VAR
	_config: INT;
END_VAR
IF Execute THEN	
	_logger.Information(_message.Reset().Append('ChuckInLoadingPosition: ').Append(TO_STRING(LoadingPosition)).ToString());
	
	IsInLoadingPosition := LoadingPosition;
	_chuckInLoadingPositionCmd := FALSE;
END_IF
END_METHOD

PROPERTY DeviceID : STRING
GET
DeviceID := _deviceID;
END_GET
SET
_deviceID := DeviceID;
END_SET
END_PROPERTY

PROPERTY Family : DeviceFamily
GET
Family := _family;
END_GET
SET
_family := Family;
END_SET
END_PROPERTY

METHOD PROTECTED IsAlive
VAR_INPUT
END_VAR
_notifyIsAlive := TRUE;

IF _lifeTimeCount < 5 THEN
	_lifeTimeCount := _lifeTimeCount + 1;
ELSE
	_lifeTimeCount := 1;
END_IF
END_METHOD

METHOD MessageSchedulerBase
VAR_INPUT
END_VAR
IF _pulseGeneratorBase.Q THEN
	_pulseGeneratorBase(IN := FALSE, PT := T#10MS);
		
	CASE _itemSchedulerBase OF			
		0:  _deliverMessagesBase := EFeedbackMsgChuckBase.IsInLoadingPositionMsg;
			ioMessage := ' ';
			_itemSchedulerBase := 1;
			
		1: _deliverMessagesBase := EFeedbackMsgChuckBase.IsInLoadingPositionMsg;
			ioMessage := TO_STRING(IsInLoadingPosition);
			_itemSchedulerBase := 0;
	END_CASE
ELSE
	_pulseGeneratorBase(IN := TRUE, PT := T#100MS);		
END_IF


IF _pulseIsAliveGenerator.Q THEN
	_pulseIsAliveGenerator(IN := FALSE, PT := T#10MS);
		
	IsAlive();	
ELSE
	_pulseIsAliveGenerator(IN := TRUE, PT := T#1000MS);		
END_IF
END_METHOD

PROPERTY Name : STRING
GET
Name := _name;
END_GET
SET
_name := Name;
END_SET
END_PROPERTY

PROPERTY WaferSize : EWaferSize
GET
WaferSize := _waferSize;
END_GET
SET
_waferSize := WaferSize;
END_SET
END_PROPERTY

END_FUNCTION_BLOCK

// ---- PMShared/Hardware/Devices/Ffus/Astrofan/Astrofan612Ffu.TcPOU
{attribute 'OPC.UA.DA' := '1'}
FUNCTION_BLOCK Astrofan612Ffu EXTENDS FfuBase
VAR
	{attribute 'OPC.UA.DA' := '0'}
	_master : ModbusRtuMasterV2_KL6x22B;
	{attribute 'OPC.UA.DA' := '0'}
	_modbusErrorId : MODBUS_ERRORS;
	{attribute 'OPC.UA.DA' := '0'}
	Quantity : WORD := 1;
	{attribute 'OPC.UA.DA' := '0'}
	Id : BYTE := 1;
	{attribute 'OPC.UA.DA' := '0'}
	_config : Astrofan612FfuConfig;		
	{attribute 'OPC.UA.DA' := '0'}
	_deliverMessages : INT;
	
	StateMsg : STRING(255);
	IsAliveMsg : STRING(255);
	CurrentSpeedMsg : STRING(255);
	TemperatureMsg : STRING(255);
	WarningRaisedMsg : STRING(255) := BOOL_TO_STRING(FALSE);
	AlarmRaisedMsg : STRING(255) := BOOL_TO_STRING(FALSE);
	CustomMsg : STRING(255);
	
	{region 'Commands'}
	{attribute 'OPC.UA.DA' := '0'}
	_powerOn : BOOL;
	{attribute 'OPC.UA.DA' := '0'}
	_powerOff : BOOL;
	{attribute 'OPC.UA.DA' := '0'}
	_customCmd : BOOL;
	{attribute 'OPC.UA.DA' := '0'}			  		   
	_raisePropertiesCmd : BOOL;
	{attribute 'OPC.UA.DA' := '0'}
	_cmd : STRING;	 
	{endregion}		
	{attribute 'OPC.UA.DA' := '0'}
	_initDevice : BOOL;	
	{attribute 'OPC.UA.DA' := '0'}
	_itemScheduler : INT;	
	{attribute 'OPC.UA.DA' := '0'}
	_pulseGenerator : TON;	
	{attribute 'OPC.UA.DA' := '0'}
	_pulseTimeout : TON;		
	{attribute 'OPC.UA.DA' := '0'}
	_itemRaisedProperties : INT;	
	{attribute 'OPC.UA.DA' := '0'}
	_pulseIsAliveGenerator : TON;	
	{attribute 'OPC.UA.DA' := '0'}
	_execPulseGenerator : TON;
	{attribute 'OPC.UA.DA' := '0'}
	_pulseLoop : TON;
	{attribute 'OPC.UA.DA' := '0'}	
	_itemSubScheduler : INT;
	{attribute 'OPC.UA.DA' := '0'}
	_itemExecScheduler : INT;
	{attribute 'OPC.UA.DA' := '0'}
	_itemSubRaisedProperties : INT;
	{attribute 'OPC.UA.DA' := '0'}
	_itemFanSpeed : INT;
	{attribute 'OPC.UA.DA' := '0'}
	message : STRING;
	{attribute 'OPC.UA.DA' := '0'}
	_lifeTimeCount : UINT;
	{attribute 'OPC.UA.DA' := '0'}
	_notifyIsAlive : BOOL;
	{attribute 'OPC.UA.DA' := '0'}
	_readData : UINT;
	{attribute 'OPC.UA.DA' := '0'}
	_readHoldingData : UINT;
	{attribute 'OPC.UA.DA' := '0'}
	_writeData : UINT;
	{attribute 'OPC.UA.DA' := '0'}
	_cmdReadInput : BOOL;
	{attribute 'OPC.UA.DA' := '0'}
	_cmdReadHolding : BOOL;
	{attribute 'OPC.UA.DA' := '0'}
	_cmdWriteSingleRegister : BOOL;
	{attribute 'OPC.UA.DA' := '0'}
	_addressInput : STRING;
	{attribute 'OPC.UA.DA' := '0'}
	_addressHolding : STRING;
	{attribute 'OPC.UA.DA' := '0'}
	_addressWrite : STRING;
	{attribute 'OPC.UA.DA' := '0'}
	_currentSpeedPercent : UINT;
	{attribute 'OPC.UA.DA' := '0'}	
	_temperature : UINT;
	{attribute 'OPC.UA.DA' := '0'}
	_maxSpeed : UINT;
	{attribute 'OPC.UA.DA' := '0'}
	_setSpeedCmd : BOOL;
	{attribute 'OPC.UA.DA' := '0'}
	_fanMaxSpeedCmd : BOOL;
	{attribute 'OPC.UA.DA' := '0'}
	_fanActualSpeedCmd : BOOL;
    {attribute 'OPC.UA.DA' := '0'}
	_setSpeedPercent : UINT;
	{attribute 'OPC.UA.DA' := '0'}
	_doneScheduler : BOOL;
	{attribute 'OPC.UA.DA' := '0'}
	_doneRaised : BOOL;
	{attribute 'OPC.UA.DA' := '0'}	
	_pressure AT %I* : UINT;
	{attribute 'OPC.UA.DA' := '0'}		
	_alarmRaised : EventRaised;
	{attribute 'OPC.UA.DA' := '0'}			
	_warningRaised : EventRaised;
END_VAR

ReadInputRegister();
ReadHoldingRegister();
WriteSingleRegister();

// Init device
InitDevice();

// Check if it's still alive
IF _notifyIsAlive THEN
	IsAliveMsg := TO_STRING(_lifeTimeCount);
	_notifyIsAlive := FALSE;
END_IF

CASE _deliverMessages OF
	EFeedbackMsgAstrofan612.StateMsg :
		;
	EFeedbackMsgAstrofan612.StatusMsg :
		;
	EFeedbackMsgAstrofan612.CurrentSpeedMsg :
		CurrentSpeedMsg := TO_STRING(_currentSpeedPercent);
	EFeedbackMsgAstrofan612.TemperatureMsg :
		TemperatureMsg := TO_STRING(_temperature);
	EFeedbackMsgAstrofan612.WarningRaisedMsg :
		;
	EFeedbackMsgAstrofan612.AlarmRaisedMsg :
		;
	EFeedbackMsgAstrofan612.CustomMsg :
		;
END_CASE

SetSpeed(_setSpeedCmd, _setSpeedPercent);
RaisePropertiesChanged(_raisePropertiesCmd);
CustomCommand(_customCmd, _cmd);


IF _config.Loop.IsEnabled THEN
	LoopFanSpeed();
	WarningRaised();
	AlarmRaised();	
END_IF


IF (NOT _setSpeedCmd AND NOT _customCmd AND NOT _raisePropertiesCmd) THEN
	MessageScheduler();
END_IF

METHOD AlarmRaised
VAR
	alarmRaised : STRING := 'ALARM';
END_VAR
_AlarmRaised(DeviceName := THIS^._name,
				EventRaisedMsg := alarmRaised,
				EventTimerSetCriteria := _currentSpeedPercent > _config.Loop.FfuLoopAlarm.ThresholdPercent, 
				EventTimerSeconds := _config.Loop.FfuLoopAlarm.TimerSeconds,
				EventMsg => );
				
IF 	_AlarmRaised.EventMsg = alarmRaised THEN
	AlarmRaisedMsg := BOOL_TO_STRING(TRUE);
ELSE
	AlarmRaisedMsg := BOOL_TO_STRING(FALSE);
END_IF
END_METHOD

{attribute 'TcRpcEnable' := '1'}
(** Custom command **)
METHOD CustomCommand
VAR_INPUT
	Execute : BOOL;
	Cmd : STRING;
END_VAR
(*IF Execute THEN
	_logger.Information(_message.Reset(). Append(_config.Name).Append(' - Custom command : '). Append(Cmd).ToString());	
	
	_deliverMessages := EFeedbackMsgAstrofan612.CustomMsg;														
	
	_customCmd := FALSE;
END_IF*)
END_METHOD

METHOD FB_init : BOOL
VAR_INPUT
	bInitRetains : BOOL; // if TRUE, the retain variables are initialized (warm start / cold start)
	bInCopyCode : BOOL;  // if TRUE, the instance afterwards gets moved into the copy code (online change)
	Config : Astrofan612FfuConfig;
END_VAR
IF Config.IsEnabled THEN
	_config := Config;
	
	SUPER^._ffuConfig.Name := Config.Name;
	SUPER^._ffuConfig.DeviceID := Config.DeviceID;
	SUPER^._ffuConfig.IsEnabled := Config.IsEnabled;
	SUPER^._ffuConfig.LogLevel := Config.LogLevel;

	SUPER^.Name := Config.Name;
	SUPER^.DeviceID := Config.DeviceID;	
	THIS^.Family := DeviceFamily.Ffu;
		
	_Logger.Information(_message.Reset().Append('Init ').
							Append('{').Append(TO_STRING(THIS^.Family)).Append('} - ').
							Append('{').Append(TO_STRING(Config.Name)).Append('}').ToString());	
END_IF
END_METHOD

METHOD GetFanActualSpeed 
VAR
	AddressActualSpeed : STRING := '16#D010';	
	currentSpeedReal : UINT;
END_VAR
IF _pulseGenerator.Q THEN
	_pulseGenerator(IN := FALSE, PT := T#10MS);
		
	CASE _itemSubScheduler OF
		0 :	_cmdReadInput := TRUE;
			_addressInput:= AddressActualSpeed;	
			_itemSubScheduler := 1;
		
		1 : _deliverMessages := EFeedbackMsgAstrofan612.CurrentSpeedMsg;
			_currentSpeedPercent := REAL_TO_UINT (( _readData * 100.00) / 65536);
			_cmdReadInput := FALSE;
			_itemSubScheduler := 0;
			_doneScheduler := TRUE;
	END_CASE	
ELSE
	_pulseGenerator(IN := TRUE, PT := T#500MS);		
END_IF
END_METHOD

METHOD GetFanMaxSpeed 
VAR
	AddressMaxSpeed : STRING := '16#D119';
END_VAR
IF _pulseGenerator.Q THEN
		_pulseGenerator(IN := FALSE, PT := T#10MS);
			
		CASE _itemSubRaisedProperties OF
			0 :	_cmdReadHolding := TRUE;
				_addressHolding := AddressMaxSpeed;
				_itemSubRaisedProperties := 1;
			
			1 : _maxSpeed := _readHoldingData;
				_cmdReadHolding := FALSE;
				_itemSubRaisedProperties := 0;		
	
				_doneRaised := TRUE;					
		END_CASE
	ELSE
		_pulseGenerator(IN := TRUE, PT := T#500MS);		
END_IF
END_METHOD

METHOD GetFanTemperature 
VAR
	AddressTemperature : STRING := '16#D015';
END_VAR
IF _pulseGenerator.Q THEN
	_pulseGenerator(IN := FALSE, PT := T#10MS);
		
	CASE _itemSubScheduler OF
		0 :	_cmdReadInput := TRUE;
			_addressInput := AddressTemperature;
			_itemSubScheduler := 1;
		
		1 : _deliverMessages := EFeedbackMsgAstrofan612.TemperatureMsg;
			_temperature := _readData;
			_cmdReadInput := FALSE;
			_itemSubScheduler := 0;
			
			_doneScheduler:= TRUE ;			
	END_CASE	
ELSE
	_pulseGenerator(IN := TRUE, PT := T#500MS);		
END_IF
END_METHOD

METHOD InitDevice
IF NOT _initDevice THEN	
	_logger.Information(_message.Reset(). Append(_config.Name). Append(' - Init device').ToString());
	
	THIS^.SetDone();
	
	_setSpeedPercent := 50;
	_setSpeedCmd := TRUE;
	_initDevice := TRUE;	
END_IF
END_METHOD

METHOD PROTECTED IsAlive
_notifyIsAlive := TRUE;

IF _lifeTimeCount < 5 THEN
	_lifeTimeCount := _lifeTimeCount + 1;
ELSE
	_lifeTimeCount := 1;
END_IF
END_METHOD

METHOD LoopFanSpeed 
VAR_INPUT
END_VAR
VAR
	differentialPressure : UINT;
END_VAR
IF _pulseLoop.Q THEN
	_pulseLoop(IN := FALSE, PT := T#10MS);
	
	differentialPressure := (_pressure * 10)/32767;
	
	IF differentialPressure <=  _config.Loop.FfuPressureMinimumValuePa THEN
		_setSpeedPercent := TO_UINT(LIMIT (_config.Loop.FfuLoopSetSpeedLowerLimitPercent, (_setSpeedPercent + 10), 
								_config.Loop.FfuLoopSetSpeedHigherLimitPercent));
		_setSpeedCmd := TRUE;
	ELSIF differentialPressure >= _config.Loop.FfuPressureMaximumValuePa THEN
		_setSpeedPercent := TO_UINT(LIMIT (_config.Loop.FfuLoopSetSpeedLowerLimitPercent, ABS(_setSpeedPercent - 10), 
								_config.Loop.FfuLoopSetSpeedHigherLimitPercent));
		_setSpeedCmd := TRUE;
	ELSE
		_SetSpeedPercent := _config.Loop.FfuLoopStandardSetSpeed;
		_setSpeedCmd := TRUE;
	END_IF
ELSE
	_pulseLoop(IN := TRUE, PT := TO_TIME(_config.Loop.FfuLoopPressureTimerSeconds*1000));
END_IF
END_METHOD

METHOD MessageScheduler
CASE _itemScheduler OF		
	0:	GetFanTemperature();	
		IF _doneScheduler THEN 
            _itemScheduler := 1;
		END_IF		
		
	1: GetFanActualSpeed();
	    IF _doneScheduler THEN 
            _itemScheduler := 0;
		END_IF	
	
END_CASE

_doneScheduler := FALSE;
END_METHOD

{attribute 'TcRpcEnable' := '1'}
METHOD RaisePropertiesChanged
VAR_INPUT
	execute : BOOL;
END_VAR
IF execute THEN
	_raisePropertiesCmd := TRUE;
	
	IF _pulseGenerator.Q THEN
		_pulseGenerator(IN := FALSE, PT := T#10MS);
		CASE _itemRaisedProperties OF
			0:  _deliverMessages := EFeedbackMsgAstrofan612.CurrentSpeedMsg;
				_currentSpeedPercent := 0;	
				_itemRaisedProperties := 1;
						
			1:	_deliverMessages := EFeedbackMsgAstrofan612.TemperatureMsg;
				_temperature := 0;	
				_itemRaisedProperties := 10;							
			
			10: _raisePropertiesCmd := FALSE;				
				_itemRaisedProperties := 0;		
		END_CASE
	ELSE
		_pulseGenerator(IN := TRUE, PT := T#50MS);	
	END_IF
END_IF
END_METHOD

METHOD ReadHoldingRegister
_master.ReadRegs (
	UnitID:= Id,
	Quantity:= Quantity,
	MBAddr:= STRING_TO_WORD(_addressHolding),
	cbLength:= SIZEOF(_readHoldingData),  
	pMemoryAddr:= ADR(_readHoldingData),  
	AuxQuantity:= ,     
	AuxMBAddr:= , 
	AuxcbLength:= , 
	pAuxMemoryAddr:= , 
	Execute:= _cmdReadHolding,
	Timeout:= T#1S,
	BUSY=> , 
	Error=> ,
	ErrorId=> _modbusErrorId, 
	cbRead=> );
END_METHOD

METHOD ReadInputRegister
_master.ReadInputRegs(
	UnitID:= Id,        
	Quantity:= Quantity,
	MBAddr:= STRING_TO_WORD(_addressInput),   
	cbLength:= SIZEOF(_readData),  
	pMemoryAddr:= ADR(_readData),  
	AuxQuantity:= ,     
	AuxMBAddr:= , 
	AuxcbLength:= , 
	pAuxMemoryAddr:= , 
	Execute:= _cmdReadInput,
	Timeout:= T#1S,
	BUSY=> , 
	Error=> , 
	ErrorId=> _modbusErrorId, 
	cbRead=> );
END_METHOD

{attribute 'TcRpcEnable' := '1'}
METHOD PROTECTED SetSpeed 
VAR_INPUT
	execute : BOOL;
	speedPercent : UINT;
END_VAR
VAR
	addressSetSpeed : STRING := '16#D001' ;
	setSpeed: UINT;
END_VAR
IF Execute THEN	
	_setSpeedCmd := TRUE;	
	_setSpeedPercent := SpeedPercent;

	IF _execPulseGenerator.Q THEN
		_execPulseGenerator(IN := FALSE, PT := T#10MS);
			
		CASE _itemExecScheduler OF
			0: 	
				_cmdReadInput := FALSE;
				_cmdReadHolding := FALSE;	
				_cmdWriteSingleRegister := FALSE;				
				_itemExecScheduler := 1;
				
			1:	IF _config.SpeedMatrix.Enable THEN
					setSpeed := ScaleSpeed(iSpeed := _setSpeedPercent, SpeedMatrix := _config.SpeedMatrix.FfuMatrix);
				ELSE
					setSpeed := _setSpeedPercent;
				END_IF
				_writeData := ((setSpeed * 65535) / 100);
				
				 _addressWrite := AddressSetSpeed;
				 _cmdWriteSingleRegister := TRUE;
				 _itemExecScheduler := 10;				
											
			10:  _cmdWriteSingleRegister := FALSE;
				_itemExecScheduler := 11;
			
			11:	GetFanActualSpeed();
				// TODO :  intégrer une tempo pour sortir de là, en cas de problème. Pour éviter la boucle infinie
				IF _doneScheduler  THEN
					_itemExecScheduler := 50;
					_doneScheduler := FALSE;
				END_IF
				
			50:  _cmdReadInput := FALSE;				
				_setSpeedCmd := FALSE;	
				_itemExecScheduler := 0;										
		END_CASE						
	ELSE
		_execPulseGenerator(IN := TRUE, PT := T#200MS);	
	END_IF
END_IF
END_METHOD

METHOD WarningRaised 
VAR
	warningRaised : STRING := 'Warning';
END_VAR
_warningRaised(DeviceName := THIS^._name,
				EventRaisedMsg := warningRaised,
				EventTimerSetCriteria := _currentSpeedPercent > _config.Loop.FfuLoopWarning.ThresholdPercent, 
				EventTimerSeconds := _config.Loop.FfuLoopWarning.TimerSeconds,
				EventMsg => );



IF 	_warningRaised.EventMsg = warningRaised THEN
	WarningRaisedMsg :=  BOOL_TO_STRING(TRUE);
ELSE
	WarningRaisedMsg :=  BOOL_TO_STRING(FALSE);
END_IF
END_METHOD

METHOD WriteSingleRegister
_master.WriteSingleRegister (
	UnitID:= Id,        
	Quantity:= Quantity,
	MBAddr:= STRING_TO_WORD(_addressWrite),   
	cbLength:= SIZEOF(_writeData),  
	pMemoryAddr:= ADR(_writeData),  
	AuxQuantity:= ,     
	AuxMBAddr:= , 
	AuxcbLength:= , 
	pAuxMemoryAddr:= , 
	Execute:= _cmdWriteSingleRegister,
	Timeout:= T#1S,
	BUSY=> , 
	Error=> , 
	ErrorId=> _modbusErrorId, 
	cbRead=> );
END_METHOD

END_FUNCTION_BLOCK

// ---- PMShared/Hardware/Devices/Ffus/FfuBase.TcPOU
FUNCTION_BLOCK ABSTRACT FfuBase EXTENDS TExecution IMPLEMENTS IDevice
VAR_INPUT
END_VAR
VAR_OUTPUT
END_VAR
VAR
	{attribute 'OPC.UA.DA' := '0'}
	_name : STRING;
	{attribute 'OPC.UA.DA' := '0'}
	_deviceID : STRING;				
	{attribute 'OPC.UA.DA' := '0'}	
	_family : DeviceFamily;	
	{attribute 'OPC.UA.DA' := '0'}
	_logger : Logger;
	{attribute 'OPC.UA.DA' := '0'}
	_message : StringBuilder;
	{attribute 'OPC.UA.DA' := '0'}
	_ffuConfig : DeviceConfiguration;	
END_VAR

PROPERTY DeviceID : STRING
GET
DeviceID := _deviceID;
END_GET
SET
_deviceID := DeviceID;
END_SET
END_PROPERTY

PROPERTY Family : DeviceFamily
GET
Family := _family;
END_GET
SET
_family := Family;
END_SET
END_PROPERTY

PROPERTY Name : STRING
GET
Name := _name;
END_GET
SET
_name := Name;
END_SET
END_PROPERTY

METHOD PROTECTED ABSTRACT SetSpeed
VAR_INPUT
	Execute : BOOL;
	SpeedPercent : UINT;
END_VAR
END_METHOD

END_FUNCTION_BLOCK

// ---- PMShared/Hardware/Devices/Ffus/Astrofan/Loop/EventRaise/EventRaised.TcPOU
FUNCTION_BLOCK EventRaised
VAR_INPUT
	EventRaisedMsg : STRING;
	EventTimerSeconds : UINT;
	EventTimerSetCriteria : BOOL;
	DeviceName	: STRING;
END_VAR
VAR_OUTPUT
	EventMsg : STRING;
END_VAR
VAR
	_eventtrigger : BOOL := FALSE;
	{attribute 'OPC.UA.DA' := '0'}	
	_eventRaised : BOOL;
	{attribute 'OPC.UA.DA' := '0'}	
	_eventTimeOut : TON;
	{attribute 'OPC.UA.DA' := '0'}	
	_logger : Logger;
	{attribute 'OPC.UA.DA' := '0'}
	_message : StringBuilder;
END_VAR

_eventTimeOut(IN := EventTimerSetCriteria,
			PT := TO_TIME(EventTimerSeconds*1000));
	IF _eventTimeOut.Q THEN
		_eventRaised := TRUE;
		eventMsg := EventRaisedMsg;
		IF	NOT _eventtrigger THEN
			_Logger.Information(_message.Reset().Append(eventMsg).Append(' - ').Append(DeviceName).ToString()); 
			_Eventtrigger := TRUE;
		END_IF
	ELSE
		_eventtrigger := FALSE;
		_eventRaised := FALSE;
		eventMsg := '';
	END_IF

END_FUNCTION_BLOCK

// ---- PMShared/Hardware/Devices/Ffus/Astrofan/Loop/FfuSpeedMatrix/ScaleSpeed.TcPOU
FUNCTION ScaleSpeed : UINT
VAR_INPUT
	iSpeed : UINT;
	SpeedMatrix	: ARRAY[0..Constants.speedMatrixSize] OF FfuSpeed;
END_VAR
VAR
	i : UINT;
	found	: BOOL := FALSE;
END_VAR

FOR i:= 1 TO Constants.speedMatrixSize DO
	IF (SpeedMatrix[i].NonScaledSpeedValue = iSpeed) THEN
		ScaleSpeed := SpeedMatrix[i].ScaledSpeedValue;
		found := TRUE;
	EXIT;
	END_IF
END_FOR

IF NOT found THEN
	ScaleSpeed := 0;
END_IF

END_FUNCTION

// ---- PMShared/Hardware/Devices/Screens/Densitron/DM430GNS/DM430GNScreenFS.TcPOU
{attribute 'OPC.UA.DA' := '1'}
FUNCTION_BLOCK DM430GNScreenFS EXTENDS DM430GNScreen
VAR_INPUT
END_VAR
VAR_OUTPUT
END_VAR
VAR
	{attribute 'OPC.UA.DA' := '0'}
	_config : DM430GNScreenConfig;
	{attribute 'OPC.UA.DA' := '0'}
	_coeAccess : CoeAccess;
	{attribute 'OPC.UA.DA' := '0'}
	_initConfigSerialCom : BOOL;
	{attribute 'OPC.UA.DA' := '0'}	
	_serialCom  : SerialCom(Prefix :='', Suffix := Const.CARRIAGE_RETURN);
	{attribute 'OPC.UA.DA' := '0'}
	_refSerialCom : REFERENCE TO SerialCom(Prefix :='', Suffix := Const.CARRIAGE_RETURN) := _serialCom;	
	
	{attribute 'OPC.UA.DA' := '0'}
	_pulseGeneratorInit : TON;	
	{attribute 'OPC.UA.DA' := '0'}
	_itemInit : INT;
END_VAR

IF _config.IsSimulated THEN
	SUPER^(Conf := _config, SerialCom := _serialCom, RefSerialCom := _refSerialCom);
ELSE
	IF NOT InitConfigSerialCom THEN
		ConfigureSerialCom();
	ELSIF THIS^.Status = TExecutionState.Ready THEN
		IF _refSerialCom.ErrorReceiveId = COMERROR_NOERROR THEN
			_refSerialCom(TxBuffer:= HardwareGlobalVariables.TxBufferDM430GNScreenFS, 
						  RxBuffer:= HardwareGlobalVariables.RxBufferDM430GNScreenFS);
		END_IF						  			
					
		SUPER^(Conf := _config, SerialCom := _serialCom, RefSerialCom := _refSerialCom);

		// Init device
		InitDevice(); 			
	END_IF
END_IF

METHOD ConfigureSerialCom
VAR_INPUT
END_VAR

VAR
	Status: INT;
END_VAR
IF _coeAccess.CoeOperation.Ready THEN
	_logger.Information(_message.Reset().Append('Start configuration com serial').ToString());
END_IF;	

_coeAccess.CoeOperation.Start();
_coeAccess(SerialCommunication := _config.SerialCommunication);
	
IF _coeAccess.CoeOperation.Done THEN
	_coeAccess.SetDone();
	
	_Logger.Information(_message.Reset().
							Append('{').Append(TO_STRING(THIS^.Family)).Append('} : ').
							Append(' - Status : ').Append(TO_STRING(_coeAccess.Status)).ToString());
	InitConfigSerialCom := TRUE;
END_IF
 
IF _coeAccess.CoeOperation.Error THEN	
	_coeAccess.SetError(0);
	
	_Logger.Error(_message.Reset().
							Append('{').Append(TO_STRING(THIS^.Family)).Append('} : ').
							Append(' - Status : ').Append(TO_STRING(_coeAccess.Status)).ToString());
	InitConfigSerialCom := TRUE;
END_IF

THIS^.Status := _coeAccess.Status;
State := _coeAccess.Status;
END_METHOD

METHOD FB_init : BOOL
VAR_INPUT
	bInitRetains : BOOL; // if TRUE, the retain variables are initialized (warm start / cold start)
	bInCopyCode : BOOL;  // if TRUE, the instance afterwards gets moved into the copy code (online change)
	Config : DM430GNScreenConfig;
END_VAR
IF Config.IsEnabled THEN
	_config := Config;
	
	SUPER^._screenConfig.Name := Config.Name;
	SUPER^._screenConfig.DeviceID := Config.DeviceID;
	SUPER^._screenConfig.IsEnabled := Config.IsEnabled;
	SUPER^._screenConfig.LogLevel := Config.LogLevel;
	
	SUPER^.Name := Config.Name;
	SUPER^.DeviceID := Config.DeviceID;	
	THIS^.Family := DeviceFamily.Screen;
		
	_Logger.Information(_message.Reset().Append('Init ').
							Append('{').Append(TO_STRING(THIS^.Family)).Append('} - ').
							Append('{').Append(TO_STRING(Config.Name)).Append('}').ToString());																													
END_IF
END_METHOD

PROPERTY InitConfigSerialCom : BOOL
GET
InitConfigSerialCom := _initConfigSerialCom;
END_GET
SET
_initConfigSerialCom := InitConfigSerialCom;
END_SET
END_PROPERTY

METHOD InitDevice
VAR_INPUT
END_VAR
VAR	
END_VAR
IF NOT _initDevice THEN		
	IF _pulseGeneratorInit.Q THEN
		_pulseGeneratorInit(IN := FALSE, PT := T#10MS);
			
		CASE _itemInit OF
			0:  _logger.Information(_message.Reset().Append(_config.Name).Append(' - Start to on').ToString());		
				_itemInit := 1;
				
			1:  _initDevice := TRUE;
				_itemInit := 0;
		END_CASE
	ELSE
		_pulseGeneratorInit(IN := TRUE, PT := T#500MS);	
	END_IF
END_IF
END_METHOD

END_FUNCTION_BLOCK

// ---- PMShared/Hardware/Devices/Screens/Densitron/DM430GNScreen.TcPOU
{attribute 'OPC.UA.DA' := '1'}
FUNCTION_BLOCK DM430GNScreen EXTENDS ScreenBase
VAR_INPUT	
	{attribute 'OPC.UA.DA' := '0'}
	Conf : DM430GNScreenConfig;		
	{attribute 'OPC.UA.DA' := '0'}
	SerialCom  : SerialCom(Prefix :='', Suffix := Const.CARRIAGE_RETURN);
	{attribute 'OPC.UA.DA' := '0'}
	RefSerialCom : REFERENCE TO SerialCom(Prefix :='', Suffix := Const.CARRIAGE_RETURN) := SerialCom;	
END_VAR
VAR_OUTPUT
END_VAR
VAR	
	{attribute 'OPC.UA.DA' := '0'}
	_deliverMessages : INT;
	
	StateMsg : STRING(255);
	StatusMsg : STRING(255);
	IsAliveMsg : STRING(255);
	PowerStateMsg : STRING(255);
	BacklightMsg : STRING(255);
	BrightnessMsg : STRING(255);
	ContrastMsg : STRING(255);
	FanAutoMsg : STRING(255);
	FanStepMsg : STRING(255);
	FanRpmMsg : STRING(255);
	TemperatureMsg : STRING(255);	
	CustomMsg : STRING(255);
	
	{region 'Commands'}
	
	{attribute 'OPC.UA.DA' := '0'}
	_powerOn : BOOL;
	{attribute 'OPC.UA.DA' := '0'}
	_powerOff : BOOL;
	
	{attribute 'OPC.UA.DA' := '0'}
	_backlight : BOOL;
	{attribute 'OPC.UA.DA' := '0'}
	_brightness : BOOL;
	{attribute 'OPC.UA.DA' := '0'}
	_contrast : BOOL;
	{attribute 'OPC.UA.DA' := '0'}
	_defaultValue : BOOL;
	{attribute 'OPC.UA.DA' := '0'}
	_fanStep : BOOL;
	{attribute 'OPC.UA.DA' := '0'}
	_sharpness : BOOL;
	{attribute 'OPC.UA.DA' := '0'}
	_fanAuto : BOOL;
	{attribute 'OPC.UA.DA' := '0'}
	_fanAutoOnCmd : BOOL;
	{attribute 'OPC.UA.DA' := '0'}
	_customCmd : BOOL;
	{attribute 'OPC.UA.DA' := '0'}			  		   
	_raiseProperties : BOOL;
	{attribute 'OPC.UA.DA' := '0'}	 
	_restoreParameters : BOOL;
	{attribute 'OPC.UA.DA' := '0'}
	_cmd : STRING;
	{attribute 'OPC.UA.DA' := '0'}
	_screenOn : BOOL;
	{attribute 'OPC.UA.DA' := '0'}
	_setBacklight : UINT;
	{attribute 'OPC.UA.DA' := '0'}
	_setBrightness : UINT;
	{attribute 'OPC.UA.DA' := '0'}
	_setContrast : UINT;
	{attribute 'OPC.UA.DA' := '0'}
	_setFanStep : EDisplayControlStep;	
	{attribute 'OPC.UA.DA' := '0'}
	_setSharpness : EDisplayControlStep;		
	{attribute 'OPC.UA.DA' := '0'}
	_ioRelayActivated : BOOL; 
				   
	{attribute 'OPC.UA.DA' := '0'}
	_screenSide : STRING;
	{attribute 'OPC.UA.DA' := '0'}
	_side : STRING;
	{attribute 'OPC.UA.DA' := '0'}
	_delimeter : STRING := ';';
		 
	{endregion}		

	{attribute 'OPC.UA.DA' := '0'}
	_initDevice : BOOL;	
	
	{attribute 'OPC.UA.DA' := '0'}
	_itemScheduler : INT;	
	{attribute 'OPC.UA.DA' := '0'}
	_pulseGenerator : TON;	
	{attribute 'OPC.UA.DA' := '0'}
	_pulseTimeout : TON;			
	{attribute 'OPC.UA.DA' := '0'}
	_itemRaisedProperties : INT;
	{attribute 'OPC.UA.DA' := '0'}
	_itemRestoreParameters : INT;	
	{attribute 'OPC.UA.DA' := '0'}
	_pulseIsAliveGenerator : TON;
	{attribute 'OPC.UA.DA' := '0'}
	_execPulseGenerator : TON;		
	{attribute 'OPC.UA.DA' := '0'}
	_execItemScheduler : INT;
	
	{attribute 'OPC.UA.DA' := '0'}
	message : STRING;
	
	{attribute 'OPC.UA.DA' := '0'}
	_lifeTimeCount : UINT;
	{attribute 'OPC.UA.DA' := '0'}
	_notifyIsAlive : BOOL;
END_VAR

IF SerialCom.ErrorSendId <> COMERROR_NOERROR THEN
	RETURN;
END_IF 

// Check if it's still alive	
IF _notifyIsAlive THEN
	IsAliveMsg := TO_STRING(_lifeTimeCount);
	_notifyIsAlive := FALSE;
END_IF

// Deliver messages
IF RefSerialCom.IsReceived THEN
	IF (Conf.DeviceID = TO_STRING(EScreenSide.Front)) THEN
		_screenSide := TO_STRING(EScreenSide.Front);
	ELSE
		_screenSide := TO_STRING(EScreenSide.Back);
	END_IF
	
	_side := CONCAT(_screenSide, _delimeter);
	message := RefSerialCom.LastReceivedString;
	
	CASE _deliverMessages OF		
		EFeedbackMsgDM430GN.StateMsg :
			;			
		EFeedbackMsgDM430GN.StatusMsg :
			;			
		EFeedbackMsgDM430GN.PowerStateMsg :
			PowerStateMsg := CONCAT(_side, ExtractMessage(message));		
		EFeedbackMsgDM430GN.BacklightMsg :
			BacklightMsg := CONCAT(_side, ExtractMessage(message));
		EFeedbackMsgDM430GN.BrightnessMsg :
			BrightnessMsg := CONCAT(_side, ExtractMessage(message));
		EFeedbackMsgDM430GN.ContrastMsg :
			ContrastMsg := CONCAT(_side, ExtractMessage(message));
		EFeedbackMsgDM430GN.FanAutoMsg :
			FanAutoMsg := CONCAT(_side, ExtractMessage(message));
		EFeedbackMsgDM430GN.FanStepMsg :
			FanStepMsg := CONCAT(_side, ExtractMessage(message));
		EFeedbackMsgDM430GN.FanRpmMsg :
			FanRpmMsg := CONCAT(_side, ExtractMessage(message));
		EFeedbackMsgDM430GN.TemperatureMsg :
			TemperatureMsg := CONCAT(_side, ExtractMessage(message));
		EFeedbackMsgDM430GN.CustomMsg :
			CustomMsg := CONCAT(_side, ExtractMessage(message));
	END_CASE	
END_IF						   							   		
	
PowerOn(_powerOn);
PowerOff(_powerOff);
SetBacklight(_backlight, _setBacklight);
SetBrightness(_brightness, _setBrightness);
SetContrast(_contrast, _setContrast);
SetDefaultValue(_defaultValue);
SetFanStep(_fanStep, _setFanStep);
SetSharpness(_sharpness, _setSharpness);
FanAutoOn(_fanAuto, _fanAutoOnCmd);
CustomCommand(_customCmd, _cmd);
RaisePropertiesChanged(_raiseProperties);	
RestoreParameters(_restoreParameters, _screenOn, _setBacklight, _setBrightness, _setContrast, _setSharpness);

IF (NOT _powerOn AND NOT _powerOff AND NOT _backlight AND NOT _brightness AND NOT _contrast AND NOT _defaultValue
 	AND NOT _fanStep AND NOT _sharpness AND NOT _fanAuto AND NOT _customCmd AND NOT _raiseProperties AND NOT _restoreParameters) THEN	
	MessageScheduler();	
END_IF

METHOD PRIVATE ConvertDecString : STRING
VAR_INPUT
	Cmd : STRING;
	Value : BYTE;
END_VAR
VAR
	tmp : STRING; 	
END_VAR

tmp := BYTE_TO_STRING(Value);
IF LEN(tmp) = 1 THEN
	tmp := BYTE_TO_DECSTR(Value, 3);
ELSIF LEN(tmp) = 2 THEN
	tmp := BYTE_TO_DECSTR(Value, 3);				
END_IF

ConvertDecString := CONCAT(cmd, tmp);
END_METHOD

{attribute 'TcRpcEnable' := '1'}
(** Custom command **)
METHOD CustomCommand
VAR_INPUT
	Execute : BOOL;
	Cmd : STRING;
END_VAR
VAR
END_VAR
IF Execute THEN
	_logger.Information(_message.Reset().Append(Conf.Name).Append(' - Custom command : ').Append(Cmd).ToString());	
	_deliverMessages := EFeedbackMsgDM430GN.CustomMsg;	
	
	SerialCom.Send(Cmd);
	_customCmd := FALSE;
END_IF
END_METHOD

METHOD PRIVATE ExtractMessage : STRING
VAR_INPUT
	Data : STRING;
END_VAR
VAR
	separator : STRING(3) := ' = ';
	split : ARRAY[0..1] OF STRING(255);
	resultSplit : BOOL;	
END_VAR

resultSplit := FindAndSplit(pSeparator := ADR(separator), pSrcString := ADR(RefSerialCom.LastReceivedString), 
                            pLeftString := ADR(split[0]), nLeftSize := SIZEOF(split[0]), 
                            pRightString := ADR(split[1]), nRightSize := SIZEOF(split[1]),
                            bSearchFromRight := FALSE );
IF resultSplit THEN
	ExtractMessage := DELETE(split[1], 1, LEN(split[1]));
ELSE	
	ExtractMessage := DELETE(RefSerialCom.LastReceivedString, 1, LEN(RefSerialCom.LastReceivedString));
END_IF
END_METHOD

{attribute 'TcRpcEnable' := '1'}
METHOD PROTECTED FanAutoOn
VAR_INPUT
	Execute : BOOL;
	AutoOn : BOOL; //0: OFF, 1: ON
END_VAR
VAR
	fanAuto : STRING;
	cmd : STRING := '000FA';
	mode : STRING;
END_VAR
IF Execute THEN	
	_fanAuto:= TRUE;	
	
	CASE _itemScheduler OF
		0:  IF AutoOn THEN
				fanAuto := 'N'; // N
				mode := 'ON';
			ELSE
				fanAuto := 'F'; // F
				mode := 'OFF';
			END_IF	
	
			_logger.Information(_message.Reset().Append(Conf.Name).Append(' - FanAutoOn: ').Append(mode).ToString());			
			SerialCom.Send(CONCAT(cmd, fanAuto)); 			
			_itemScheduler := 1;
		
		1:  GetFanAuto();				
			_fanAuto := FALSE;	
			_itemScheduler := 0;							
	END_CASE
	
	
END_IF
END_METHOD

METHOD PROTECTED GetBacklight 
VAR_INPUT
END_VAR
VAR
	cmd : STRING := '000GKV';
END_VAR
_deliverMessages := EFeedbackMsgDM430GN.BacklightMsg;
SerialCom.Send(cmd);
END_METHOD

METHOD PROTECTED GetBrightness 
VAR_INPUT
END_VAR
VAR
	cmd : STRING := '000GBV'; 
END_VAR
_deliverMessages := EFeedbackMsgDM430GN.BrightnessMsg;
SerialCom.Send(cmd);
END_METHOD

METHOD PROTECTED GetContrast 
VAR_INPUT
END_VAR
VAR
	cmd : STRING := '000GCV';
END_VAR
_deliverMessages := EFeedbackMsgDM430GN.ContrastMsg;
SerialCom.Send(cmd);
END_METHOD

METHOD PROTECTED GetFanAuto 
VAR_INPUT
END_VAR
VAR
	cmd : STRING := '000GFA'; 
END_VAR
_deliverMessages := EFeedbackMsgDM430GN.FanAutoMsg;
SerialCom.Send(cmd);
END_METHOD

METHOD PROTECTED GetFanRpm 
VAR_INPUT
END_VAR
VAR
	cmd : STRING := '000GFR';
END_VAR
_deliverMessages := EFeedbackMsgDM430GN.FanRpmMsg;
SerialCom.Send(cmd);
END_METHOD

METHOD PROTECTED GetFanStep 
VAR_INPUT
END_VAR
VAR
	cmd : STRING := '000GFV'; 
END_VAR
_deliverMessages := EFeedbackMsgDM430GN.FanStepMsg;
SerialCom.Send(cmd);
END_METHOD

METHOD PROTECTED GetPowerState 
VAR_INPUT
END_VAR
VAR 
	cmd : STRING := '000GPV';
END_VAR
_deliverMessages := EFeedbackMsgDM430GN.PowerStateMsg;
SerialCom.Send(cmd);
END_METHOD

METHOD PROTECTED GetTemperature 
VAR_INPUT
END_VAR
VAR
	cmd : STRING := '000GTV';
END_VAR
_deliverMessages := EFeedbackMsgDM430GN.TemperatureMsg;
SerialCom.Send(cmd);
END_METHOD

METHOD InitDevice
VAR_INPUT
END_VAR
IF NOT _initDevice THEN	
	_logger.Information(_message.Reset(). Append(Conf.Name). Append(' - Init device').ToString());
	
	THIS^.SetDone();
	_initDevice := TRUE;	
END_IF
END_METHOD

METHOD PROTECTED IsAlive
VAR_INPUT
END_VAR
_notifyIsAlive := TRUE;

IF _lifeTimeCount < 5 THEN
	_lifeTimeCount := _lifeTimeCount + 1;
ELSE
	_lifeTimeCount := 1;
END_IF
END_METHOD

METHOD MessageScheduler
VAR_INPUT
END_VAR
IF _pulseGenerator.Q THEN
	_pulseGenerator(IN := FALSE, PT := T#10MS);
	
	CASE _itemScheduler OF					
		0:	GetTemperature(); 
			_itemScheduler := 1;

		1:	GetPowerState(); 
			_itemScheduler := 0;	

	END_CASE
ELSE
	_pulseGenerator(IN := TRUE, PT := T#2000MS);		
END_IF



IF _pulseIsAliveGenerator.Q THEN
	_pulseIsAliveGenerator(IN := FALSE, PT := T#10MS);
		
	IsAlive();	
ELSE
	_pulseIsAliveGenerator(IN := TRUE, PT := T#1000MS);		
END_IF
END_METHOD

{attribute 'TcRpcEnable' := '1'}
METHOD PROTECTED PowerOff
VAR_INPUT
	Execute : BOOL;
END_VAR
VAR
	cmd : STRING := '000KPF'; 
END_VAR
IF Execute THEN	
	_logger.Information(_message.Reset().Append(Conf.Name).Append(' - PowerOff').ToString());
	SerialCom.Send(cmd);
	
	_powerOff := FALSE;
END_IF
END_METHOD

{attribute 'TcRpcEnable' := '1'}
METHOD PROTECTED PowerOn
VAR_INPUT
	Execute : BOOL;
END_VAR
VAR 
	cmd : STRING := '000KPN';
END_VAR
IF Execute THEN	
	_powerOn := TRUE;	
	
	IF _execPulseGenerator.Q THEN
		_execPulseGenerator(IN := FALSE, PT := T#10MS);
		CASE _execItemScheduler OF
			0: _logger.Information(_message.Reset().Append(Conf.Name).Append(' - PowerOn').ToString());
				SerialCom.Send(cmd);
				
				_execItemScheduler := 1;
			
			1:  GetPowerState();
				_execItemScheduler := 2;
	
			2:	_powerOn := FALSE;
				_execItemScheduler := 0;							
		END_CASE
	ELSE
		_execPulseGenerator(IN := TRUE, PT := T#400MS);	
	END_IF		
END_IF
END_METHOD

{attribute 'TcRpcEnable' := '1'}
METHOD RaisePropertiesChanged
VAR_INPUT
	Execute : BOOL;
END_VAR
IF Execute THEN		
	_raiseProperties := TRUE;	
	
	IF _pulseGenerator.Q THEN
		_pulseGenerator(IN := FALSE, PT := T#10MS);
		
		CASE _itemRaisedProperties OF		
			0:  StateMsg := ' ';
				StatusMsg := ' ';
				BacklightMsg := ' ';
				BrightnessMsg := ' ';
				ContrastMsg := ' ';
				FanAutoMsg := ' ';				
				FanStepMsg := ' ';
				FanRpmMsg := ' ';				
				CustomMsg := ' ';
				
				_itemRaisedProperties := 10;											
			
			10 : GetBacklight();
				 _itemRaisedProperties := 11;
				 
			11 : GetBrightness();
				 _itemRaisedProperties := 12;
				 
			12 : GetContrast();
				 _itemRaisedProperties := 13;
				 
			13 : GetFanAuto();
				 _itemRaisedProperties := 14;
				
			14 : GetFanRpm();
				_itemRaisedProperties := 15;
				
			15:  GetFanStep();
				_itemRaisedProperties := 16;				
							
			16:  _logger.Information(_message.Reset().Append(Conf.Name).Append(' - RaisePropertiesChanged').ToString());
				_raiseProperties := FALSE;				
				_itemRaisedProperties := 0;
		END_CASE
	
	ELSE
		_pulseGenerator(IN := TRUE, PT := T#200MS);	
	END_IF		
END_IF
END_METHOD

{attribute 'TcRpcEnable' := '1'}
METHOD RestoreParameters	
VAR_INPUT
	Execute : BOOL;
	ScreenOn : BOOL; 
	BacklightValue : UINT;
	BrightnessValue : UINT;
	ContrastValue : UINT;
	SharpnessValue : EDisplayControlStep;
END_VAR
IF Execute THEN		
	_restoreParameters := TRUE;	
	
	CASE _itemRestoreParameters OF		
		0:  _logger.Information(_message.Reset().Append(Conf.Name).Append(' - Start RestoreParameters').ToString());
			_itemRestoreParameters := 10;	
	
		10:  _powerOn := TRUE;
			IF NOT _powerOn THEN
				_itemRestoreParameters := 11;
			END_IF																		
		
		11 : _backlight := TRUE;
			_setBacklight := BacklightValue;
			
			IF NOT _backlight THEN
				_itemRestoreParameters := 12;
			END_IF
			 
		12 : _brightness := TRUE;
			_setBrightness := BrightnessValue;
    
			IF NOT _brightness THEN
				_itemRestoreParameters := 13;
			END_IF
			 
		13 : _contrast := TRUE;
			_setContrast := ContrastValue;
    
			IF NOT _contrast THEN
				_itemRestoreParameters := 14;
			END_IF
			 
		14 : _sharpness := TRUE;
			_setSharpness := SharpnessValue;
    
			IF NOT _sharpness THEN
				_itemRestoreParameters := 20;
			END_IF													
						
		20:  _logger.Information(_message.Reset().Append(Conf.Name).Append(' - Finish RestoreParameters').ToString());
			_restoreParameters := FALSE;				
			_itemRestoreParameters := 0;
	END_CASE		
END_IF
END_METHOD

{attribute 'TcRpcEnable' := '1'}
METHOD PROTECTED SetBacklight
VAR_INPUT
	Execute : BOOL;
	Value : UINT;
END_VAR
VAR	
	cmd : STRING := '000SKV';
END_VAR
IF Execute THEN	
	_backlight := TRUE;	
	_setBacklight := Value;
	
	IF _execPulseGenerator.Q THEN
		_execPulseGenerator(IN := FALSE, PT := T#10MS);
		CASE _execItemScheduler OF
			0:  IF _setBacklight >= 0 OR _setBacklight <= 100 THEN
					_logger.Information(_message.Reset().Append(Conf.Name).Append(' - SetBacklight: ').Append(TO_STRING(_setBacklight)).ToString());																	
					SerialCom.Send(ConvertDecString(cmd, UINT_TO_BYTE(_setBacklight)));					
				ELSE
					_logger.Error(_message.Reset().Append(Conf.Name).Append(' - SetBacklight - Out of range : ').Append(TO_STRING(_setBacklight)).ToString());				
				END_IF
				
				_execItemScheduler := 1;
			
			1:  GetBacklight();
				_execItemScheduler := 2;
	
			2:	_backlight := FALSE;	
				_execItemScheduler := 0;							
		END_CASE
	ELSE
		_execPulseGenerator(IN := TRUE, PT := T#400MS);	
	END_IF										
END_IF
END_METHOD

{attribute 'TcRpcEnable' := '1'}
METHOD PROTECTED SetBrightness
VAR_INPUT
	Execute : BOOL;
	Value : UINT;
END_VAR
VAR
	cmd : STRING := '000SBV';
END_VAR
IF Execute THEN	
	_brightness := TRUE;
	
	_setBrightness := Value;
	
	IF _execPulseGenerator.Q THEN
		_execPulseGenerator(IN := FALSE, PT := T#10MS);
		CASE _execItemScheduler OF
			0:  IF _setBrightness >= 0 OR _setBrightness <= 100 THEN
					_logger.Information(_message.Reset().Append(Conf.Name).Append(' - SetBrightness: ').Append(TO_STRING(_setBrightness)).ToString());									
					SerialCom.Send(ConvertDecString(cmd, UINT_TO_BYTE(_setBrightness)));					
				ELSE
					_logger.Error(_message.Reset().Append(Conf.Name).Append(' - SetBrightness - Out of range : ').Append(TO_STRING(_setBrightness)).ToString());
				END_IF
				
				_execItemScheduler := 1;
			
			1:  GetBrightness();
				_execItemScheduler := 2;
				
			2:	_brightness := FALSE;	
				_execItemScheduler := 0;							
		END_CASE
	ELSE
		_execPulseGenerator(IN := TRUE, PT := T#400MS);	
	END_IF										
END_IF
END_METHOD

{attribute 'TcRpcEnable' := '1'}
METHOD PROTECTED SetContrast
VAR_INPUT
	Execute : BOOL;
	Value : UINT;
END_VAR
VAR
	cmd : STRING := '000SCV';
	tmp : STRING;
END_VAR
IF Execute THEN	
	_contrast := TRUE;
	_setContrast := Value;
	
	IF _execPulseGenerator.Q THEN
		_execPulseGenerator(IN := FALSE, PT := T#10MS);
		CASE _execItemScheduler OF
			0:  IF _setContrast >= 0 OR _setContrast <= 100 THEN
					_logger.Information(_message.Reset().Append(Conf.Name).Append(' - SetContrast: ').Append(TO_STRING(_setContrast)).ToString());													
					SerialCom.Send(ConvertDecString(cmd, UINT_TO_BYTE(_setContrast)));					
				ELSE
					_logger.Error(_message.Reset().Append(Conf.Name).Append(' - SetContrast - Out of range : ').Append(TO_STRING(_setContrast)).ToString());
				END_IF
				
				_execItemScheduler := 1;
			
			1:  GetContrast();	
				_execItemScheduler := 2;
			
			2:	_contrast := FALSE;	
				_execItemScheduler := 0;							
		END_CASE	
	ELSE
		_execPulseGenerator(IN := TRUE, PT := T#400MS);	
	END_IF								
END_IF
END_METHOD

{attribute 'TcRpcEnable' := '1'}
METHOD PROTECTED SetDefaultValue
VAR_INPUT
	Execute : BOOL;
END_VAR
VAR	
	cmd : STRING := '000DFT'; 
END_VAR
IF Execute THEN		
	_logger.Information(_message.Reset().Append(Conf.Name).Append(' - SetDefaultValue').ToString());	
	SerialCom.Send(cmd);	
	
	_defaultValue := FALSE;
END_IF
END_METHOD

{attribute 'TcRpcEnable' := '1'}
METHOD PROTECTED SetFanStep
VAR_INPUT
	Execute : BOOL;
	Value : EDisplayControlStep;
END_VAR
VAR
	cmd : STRING := '000SFV00';
END_VAR
IF Execute THEN	
	_fanStep := TRUE;
	_setFanStep := Value;
	
	IF _execPulseGenerator.Q THEN
		_execPulseGenerator(IN := FALSE, PT := T#10MS);
		CASE _execItemScheduler OF
			0: _logger.Information(_message.Reset().Append(Conf.Name).Append(' - SetFanStep: ').Append(TO_STRING(_setFanStep)).ToString());			
				SerialCom.Send(CONCAT(cmd, TO_STRING(_setFanStep)));				
				_execItemScheduler := 1;
			
			1:  GetFanStep();	
				_execItemScheduler := 2;
			
			2:	_fanStep := FALSE;	
				_execItemScheduler := 0;							
		END_CASE	
	ELSE
		_execPulseGenerator(IN := TRUE, PT := T#400MS);	
	END_IF						
END_IF
END_METHOD

{attribute 'TcRpcEnable' := '1'}
METHOD PROTECTED SetSharpness
VAR_INPUT
	Execute : BOOL;
	Value : EDisplayControlStep;
END_VAR
VAR
	cmd : STRING := '000SSV00';
END_VAR
IF Execute THEN		
	_sharpness := TRUE;
	_setSharpness := Value;
 
	IF _execPulseGenerator.Q THEN
		_execPulseGenerator(IN := FALSE, PT := T#10MS);
		CASE _execItemScheduler OF
			0: _logger.Information(_message.Reset().Append(Conf.Name).Append(' - SetSharpness: ').Append(TO_STRING(_setSharpness)).ToString());
				SerialCom.Send(CONCAT(cmd, TO_STRING(_setSharpness)));				
				_execItemScheduler := 1;
			
			1:  _sharpness := FALSE;
				_execItemScheduler := 0;												
		END_CASE
	ELSE
		_execPulseGenerator(IN := TRUE, PT := T#400MS);	
	END_IF
END_IF
END_METHOD

END_FUNCTION_BLOCK

// ---- PMShared/Hardware/Devices/Screens/ScreenBase.TcPOU
FUNCTION_BLOCK ScreenBase EXTENDS TExecution IMPLEMENTS IDevice
VAR_INPUT
END_VAR
VAR_OUTPUT
END_VAR
VAR
	{attribute 'OPC.UA.DA' := '0'}
	_name : STRING;
	{attribute 'OPC.UA.DA' := '0'}
	_deviceID : STRING;				
	{attribute 'OPC.UA.DA' := '0'}	
	_family : DeviceFamily;	
	{attribute 'OPC.UA.DA' := '0'}
	_logger : Logger;
	{attribute 'OPC.UA.DA' := '0'}
	_message : StringBuilder;
	{attribute 'OPC.UA.DA' := '0'}
	_screenConfig : DeviceConfiguration;	
END_VAR

PROPERTY DeviceID : STRING
GET
DeviceID := _deviceID;
END_GET
SET
_deviceID := DeviceID;
END_SET
END_PROPERTY

PROPERTY Family : DeviceFamily
GET
Family := _family;
END_GET
SET
_family := Family;
END_SET
END_PROPERTY

PROPERTY Name : STRING
GET
Name := _name;
END_GET
SET
_name := Name;
END_SET
END_PROPERTY

END_FUNCTION_BLOCK

// ---- PMShared/Hardware/Devices/Screens/Densitron/DM430GNS/DM430GNScreenBS.TcPOU
{attribute 'OPC.UA.DA' := '1'}
FUNCTION_BLOCK DM430GNScreenBS EXTENDS DM430GNScreen
VAR_INPUT
END_VAR
VAR_OUTPUT
END_VAR
VAR
	{attribute 'OPC.UA.DA' := '0'}
	_config : DM430GNScreenConfig;
	{attribute 'OPC.UA.DA' := '0'}
	_coeAccess : CoeAccess;
	{attribute 'OPC.UA.DA' := '0'}
	_initConfigSerialCom : BOOL;
	{attribute 'OPC.UA.DA' := '0'}	
	_serialCom  : SerialCom(Prefix :='', Suffix := Const.CARRIAGE_RETURN);
	{attribute 'OPC.UA.DA' := '0'}
	_refSerialCom : REFERENCE TO SerialCom(Prefix :='', Suffix := Const.CARRIAGE_RETURN) := _serialCom;	
	
	{attribute 'OPC.UA.DA' := '0'}
	_pulseGeneratorInit : TON;	
	{attribute 'OPC.UA.DA' := '0'}
	_itemInit : INT;
END_VAR

IF _config.IsSimulated THEN
	SUPER^(Conf := _config, SerialCom := _serialCom, RefSerialCom := _refSerialCom);
ELSE
	IF NOT InitConfigSerialCom THEN
		ConfigureSerialCom();
	ELSIF THIS^.Status = TExecutionState.Ready THEN
		IF _refSerialCom.ErrorReceiveId = COMERROR_NOERROR THEN
			_refSerialCom(TxBuffer:= HardwareGlobalVariables.TxBufferDM430GNScreenBS, 
						  RxBuffer:= HardwareGlobalVariables.RxBufferDM430GNScreenBS);
		END_IF						  			
					
		SUPER^(Conf := _config, SerialCom := _serialCom, RefSerialCom := _refSerialCom);

		// Init device
		InitDevice(); 			
	END_IF
END_IF

METHOD ConfigureSerialCom
VAR_INPUT
END_VAR

VAR
	Status: INT;
END_VAR
IF _coeAccess.CoeOperation.Ready THEN
	_logger.Information(_message.Reset().Append('Start configuration com serial').ToString());
END_IF;	

_coeAccess.CoeOperation.Start();
_coeAccess(SerialCommunication := _config.SerialCommunication);
	
IF _coeAccess.CoeOperation.Done THEN
	_coeAccess.SetDone();
	
	_Logger.Information(_message.Reset().
							Append('{').Append(TO_STRING(THIS^.Family)).Append('} : ').
							Append(' - Status : ').Append(TO_STRING(_coeAccess.Status)).ToString());
	InitConfigSerialCom := TRUE;
END_IF
 
IF _coeAccess.CoeOperation.Error THEN	
	_coeAccess.SetError(0);
	
	_Logger.Error(_message.Reset().
							Append('{').Append(TO_STRING(THIS^.Family)).Append('} : ').
							Append(' - Status : ').Append(TO_STRING(_coeAccess.Status)).ToString());
	InitConfigSerialCom := TRUE;
END_IF

THIS^.Status := _coeAccess.Status;
State := _coeAccess.Status;
END_METHOD

METHOD FB_init : BOOL
VAR_INPUT
	bInitRetains : BOOL; // if TRUE, the retain variables are initialized (warm start / cold start)
	bInCopyCode : BOOL;  // if TRUE, the instance afterwards gets moved into the copy code (online change)
	Config : DM430GNScreenConfig;
END_VAR
IF Config.IsEnabled THEN
	_config := Config;
	
	SUPER^._screenConfig.Name := Config.Name;
	SUPER^._screenConfig.DeviceID := Config.DeviceID;
	SUPER^._screenConfig.IsEnabled := Config.IsEnabled;
	SUPER^._screenConfig.LogLevel := Config.LogLevel;
	
	SUPER^.Name := Config.Name;
	SUPER^.DeviceID := Config.DeviceID;	
	THIS^.Family := DeviceFamily.Screen;
		
	_Logger.Information(_message.Reset().Append('Init ').
							Append('{').Append(TO_STRING(THIS^.Family)).Append('} - ').
							Append('{').Append(TO_STRING(Config.Name)).Append('}').ToString());																													
END_IF
END_METHOD

PROPERTY InitConfigSerialCom : BOOL
GET
InitConfigSerialCom := _initConfigSerialCom;
END_GET
SET
_initConfigSerialCom := InitConfigSerialCom;
END_SET
END_PROPERTY

METHOD InitDevice
VAR_INPUT
END_VAR
VAR	
END_VAR
IF NOT _initDevice THEN		
	IF _pulseGeneratorInit.Q THEN
		_pulseGeneratorInit(IN := FALSE, PT := T#10MS);
			
		CASE _itemInit OF
			0:  _logger.Information(_message.Reset().Append(_config.Name).Append(' - Start to on').ToString());		
				_itemInit := 1;
							
			1:  _initDevice := TRUE;
				_itemInit := 0;
		END_CASE
	ELSE
		_pulseGeneratorInit(IN := TRUE, PT := T#500MS);	
	END_IF
END_IF
END_METHOD

END_FUNCTION_BLOCK

// ---- PMShared/Hardware/Devices/Rfids/Balluff/BisL405Rfid.TcPOU
{attribute 'OPC.UA.DA' := '1'}
FUNCTION_BLOCK BisL405Rfid EXTENDS RfidBase
VAR_INPUT
	IoBisL405Rfid : IoBisL405Rfid;
END_VAR
VAR_OUTPUT
END_VAR
VAR
	
	{attribute 'OPC.UA.DA' := '0'}
	_config : BisL405RfidConfig;
	
	{attribute 'OPC.UA.DA' := '0'}
	_deliverMessages : INT;
	
	DataCarrierMsg : STRING(255);
	
	{attribute 'OPC.UA.DA' := '0'}
	_initDevice : BOOL;
	
	{attribute 'OPC.UA.DA' := '0'}
	_itemInit : INT;
	
	{attribute 'OPC.UA.DA' := '0'}
	_itemScheduler : INT;
	{attribute 'OPC.UA.DA' := '0'}
	_itemExecScheduler : INT;
	
	{attribute 'OPC.UA.DA' := '0'}
	_itemExecReadTag : INT; //COUNTER
	{attribute 'OPC.UA.DA' := '0'}
	_itemExecReadTagWAIT : INT; //COUNTER
	
	{region ' CONFIGURE read BEHAVIOUR TEST options'}

	{attribute 'OPC.UA.DA' := '0'}
	_iReadTagTestRereadN : INT := 0; //3; number of time to re-read tag //CONFIGURE TEST //TEST ONLY

	{endregion}

	{region ' CONFIGURE read BEHAVIOUR options'}

	{attribute 'OPC.UA.DA' := '0'}
	_iReadStepMax : INT := 40; //max ticks/steps when tag detected //CONFIGURE 
	{attribute 'OPC.UA.DA' := '0'}
	_iReadStepMaxWait : INT := 10; //max ticks/steps when tag NOT detected //CONFIGURE 
	{attribute 'OPC.UA.DA' := '0'}
	_iReadTagBadFormatRereadN : INT := 3; //number of time to re-read tag (if 'TagBadFormat') //CONFIGURE 

	{endregion}

	{region 'control ACTIONS for signal input/output'}
	
	{attribute 'OPC.UA.DA' := '0'}
	_iDoReset : INT := 3;// 1=do it, >1 = COUNTDOWN //CONFIGURE restart at start of read
	{attribute 'OPC.UA.DA' := '0'}
	_iToggleAddressCountAfterReset : INT := 1; //3;// 1=do it, >1 = COUNTDOWN //CONFIGURE ---------------------------------------
	{attribute 'OPC.UA.DA' := '0'}
	_iToggleAddressCountAfterToggle : INT := 3;// 1=do it, >1 = COUNTDOWN //CONFIGURE -------------------------------------------
	{attribute 'OPC.UA.DA' := '0'}
	_iToggleAddress : INT := 0;// 1=do it, >1 = COUNTDOWN //CONFIGURE or set after 'Reset'/'Toggle'
	
	{attribute 'OPC.UA.DA' := '0'}
	_iReadTagRetry : INT := 0; //COUNT
	{attribute 'OPC.UA.DA' := '0'}
	_iReadDone : INT := 0; //COUNT
	{attribute 'OPC.UA.DA' := '0'}
	ToggleReset : BOOL;// := FALSE;//action flag
	{attribute 'OPC.UA.DA' := '0'}
	_uBitFlagWaitOn : UINT;// bit values 1=wait next 't' on, 2=wait 'S' on, 
	
	{attribute 'OPC.UA.DA' := '0'}
	_bPrevStrobe : BOOL;//save flag
	{attribute 'OPC.UA.DA' := '0'}
	_bLatchStrobeChanged : BOOL;//detect & latch
	{attribute 'OPC.UA.DA' := '0'}
	_bLatchADRToggled : BOOL := FALSE;//detect & latch
	
	{endregion}
	
	{attribute 'OPC.UA.DA' := '0'}
	_itemRaisedProperties : INT;
	{attribute 'OPC.UA.DA' := '0'}
	_pulseGenerator : TON;
	{attribute 'OPC.UA.DA' := '0'}
	_execPulseGenerator : TON;	
	
	{region 'Commands'}
	
	{attribute 'OPC.UA.DA' := '0'}			  		   
	_readTagCmd : BOOL;
	{attribute 'OPC.UA.DA' := '0'}			  		   
	_raiseProperties : BOOL;
	
	{endregion}	
	
	{attribute 'OPC.UA.DA' := '0'}
	message : STRING;
	
	{attribute 'OPC.UA.DA' := '0'}	
	_sMsgBuild : STRING;
END_VAR


// Init device
InitDevice(); 				  				 

// Deliver messages
CASE _deliverMessages OF			
	EFeedbackMsgBisL405.DataCarrierMsg :
		IF DataCarrierMsg <> message THEN
			DataCarrierMsg := message;	
		END_IF				
END_CASE							   							   	
	
ReadTag(_readTagCmd);
RaisePropertiesChanged(_raiseProperties);

IF NOT _raiseProperties THEN
	MessageScheduler();
END_IF

METHOD FB_init : BOOL
VAR_INPUT
	bInitRetains : BOOL; // if TRUE, the retain variables are initialized (warm start / cold start)
	bInCopyCode : BOOL;  // if TRUE, the instance afterwards gets moved into the copy code (online change)
	Config : BisL405RfidConfig;
END_VAR
IF Config.IsEnabled THEN
	_config := Config;
	
	SUPER^._rfidConfig.Name := Config.Name;
	SUPER^._rfidConfig.DeviceID := Config.DeviceID;
	SUPER^._rfidConfig.IsEnabled := Config.IsEnabled;
	SUPER^._rfidConfig.LogLevel := Config.LogLevel;
	
	SUPER^.Name := Config.Name;
	SUPER^.DeviceID := Config.DeviceID;
	
	THIS^.Family := DeviceFamily.Rfid;

	THIS^.SetReady();
	_Logger.Information(_message.Reset().Append('Init ').
							Append('{').Append(TO_STRING(THIS^.Family)).Append('} - ').
							Append('{').Append(TO_STRING(THIS^.Name)).Append('} - ').
							Append('Status : ').Append(TO_STRING(THIS^.Status)).
							ToString());										 
END_IF
END_METHOD

METHOD InitDataRead : BOOL
VAR_INPUT
END_VAR
//:	_sDBMsg:= '';//TEST ONLY
message := ' '; //clear result
_sMsgBuild := ' '; //clear result build
_itemExecReadTag := 0;//Reset read data step count
_itemExecReadTagWAIT := 0;//Reset read data step count
_iDoReset := 1;//do restart before read
_iToggleAddress:= 0;//INIT: //OFF
_uBitFlagWaitOn := 0;//INIT: 'DoReset' will set to 1 to wait for 't' signal (tag present)
_bLatchStrobeChanged:=TRUE; //INIT: bStrobeChange TRUE, set true for 1st 'ToggleAddress'
_bLatchADRToggled:=FALSE; //INIT: clear
END_METHOD

METHOD InitDevice
VAR_INPUT
END_VAR
IF NOT _initDevice THEN			
	_logger.Information(_message.Reset().
								Append(_config.Name).
								Append(' - init device').ToString());		
								
	_initDevice := TRUE;
END_IF
END_METHOD

METHOD MessageScheduler
VAR_INPUT
END_VAR
IF _pulseGenerator.Q THEN
	_pulseGenerator(IN := FALSE, PT := T#10MS);
		
	CASE _itemScheduler OF	
		0:	
			_itemScheduler := 10;
			
		10 : 
			_itemScheduler := 0;											
	END_CASE
ELSE
	_pulseGenerator(IN := TRUE, PT := T#100MS);	
END_IF
END_METHOD

{attribute 'TcRpcEnable' := '1'}
METHOD RaisePropertiesChanged
VAR_INPUT
	Execute : BOOL;
END_VAR
IF Execute THEN		
	_raiseProperties := TRUE;	
	
	IF _pulseGenerator.Q THEN
		_pulseGenerator(IN := FALSE, PT := T#10MS);
		
		CASE _itemRaisedProperties OF		
			0:  _readTagCmd := TRUE;
				_itemRaisedProperties := 10;
				
			10: _logger.Information(_message.Reset().Append(_config.Name).Append(' - RaisePropertiesChanged').ToString());
				_raiseProperties := FALSE;
				_itemRaisedProperties := 0;
		
		END_CASE
	
	ELSE
		_pulseGenerator(IN := TRUE, PT := T#100MS);	
	END_IF
		
END_IF
END_METHOD

{attribute 'TcRpcEnable' := '1'}
METHOD ReadTag
VAR_INPUT
	Execute : BOOL;
END_VAR
VAR
	CombinedByte: BYTE; 
	CombinedByte1: BYTE;

	bStrobeChange : BOOL;//detect
	//
	bLatchStrobeChanged : BOOL;//detect & latch, temp local copy...
	lRand:LREAL; //EC//20240715
	
	bTagValid : BOOL;
	
	lenghtMsg : INT;
END_VAR
IF Execute THEN
	_readTagCmd := TRUE;
	
	_deliverMessages := EFeedbackMsgBisL405.DataCarrierMsg;
	
	IF _execPulseGenerator.Q THEN
		_execPulseGenerator(IN := FALSE, PT := T#100MS);
			
		CASE _itemExecScheduler OF
			0:  //init for read
				_logger.Information(_message.Reset().Append(_config.Name).Append(' - ReadTag').ToString());
				_itemExecScheduler := 1;
				InitDataRead();
				SignalClear_ADR_and_RESTART();//clear at START
			
			1:  //reset reader & read tag data, byte by byte
				IF IoBisL405Rfid.Strobe <> _bPrevStrobe THEN
					bStrobeChange:=TRUE;
				ELSE
					bStrobeChange:=FALSE;
				END_IF
				_bPrevStrobe:= IoBisL405Rfid.Strobe;
				IF bStrobeChange THEN
					_bLatchStrobeChanged:=TRUE;//reset by 'ToggleAddress' ('OUTPUT a OFF'/'OUTPUT a ON')
				END_IF

				bLatchStrobeChanged:= _bLatchStrobeChanged; //need a copy that won't be reset (by 'ToggleAddress')
					
				CombinedByte := SignalsGet_DataByte();
				CombinedByte1:= CombinedByte;
				IF IoBisL405Rfid.TagPresent AND IoBisL405Rfid.Strobe THEN
					CombinedByte1:= CombinedByte1+1;
				END_IF
				
				IF NOT Toggle_RESTART() THEN //restart if neened (at start of reading)
					IF IoBisL405Rfid.TagPresent THEN
						_uBitFlagWaitOn:= _uBitFlagWaitOn AND (NOT 1);//clear bit
					END_IF
					IF IoBisL405Rfid.Strobe THEN
						_uBitFlagWaitOn:= _uBitFlagWaitOn AND (NOT 2);//clear bit
					END_IF
					IF _uBitFlagWaitOn = 0 THEN
						Toggle_ADR();
					ELSE
						_itemExecReadTagWAIT := _itemExecReadTagWAIT+1;//COUNT step WAIT
					END_IF
				END_IF
				_itemExecReadTag := _itemExecReadTag+1;//COUNT step
				//------------------------------------------------------------------------*
				//CONCATENATE any read charcter to RESULT STRING...
				//------------------------------------------------------------------------*								
				IF IoBisL405Rfid.TagPresent AND bLatchStrobeChanged AND bStrobeChange THEN
					IF (CombinedByte > 0) THEN
						_sMsgBuild := CONCAT(_sMsgBuild, BYTE_TO_HEXSTR(CombinedByte,2,FALSE)); //<-- ADD another BYTE to read TAG DATA
					ELSE
						IF _bLatchADRToggled THEN
							_itemExecScheduler := 2;//STOP read tag DATA
						END_IF
					END_IF
				END_IF
																
				IF _itemExecReadTag >= _iReadStepMax THEN //limit
					_itemExecScheduler := 2;//STOP read tag DATA
				END_IF
				IF _itemExecReadTagWAIT >= _iReadStepMaxWait THEN //limit
					_itemExecScheduler := 2;//STOP read tag DATA
				END_IF
				
			2:  lenghtMsg := Len(_sMsgBuild);
				IF lenghtMsg = 1  THEN
					_sMsgBuild := 'Tag not present';					
				END_IF
				_itemExecScheduler := 10;//STOP read tag DATA
				
			10:  //end read, return any data
				_readTagCmd := FALSE;	
				_itemExecScheduler := 0;		
				SignalClear_ADR_and_RESTART();//clear at END
				//VALIDATE TAG DATA...
				bTagValid:= TRUE;
				IF (_sMsgBuild <> ' ') THEN
					_iReadDone := _iReadDone+1;
				END_IF
				IF LEN(_sMsgBuild) <> 7 THEN
					bTagValid:= FALSE; //7 chars expected
				END_IF
				//ADD any other validation criteria here...
				message := _sMsgBuild; 
				
				_logger.Information(_message.Reset().Append(_config.Name).Append(': ').Append(message).ToString());
				
				//TagBadFormat retry
				IF (NOT bTagValid) AND (_iReadTagBadFormatRereadN > 0) THEN
					IF _iReadTagBadFormatRereadN > _iReadTagRetry THEN
						_readTagCmd := TRUE;//retry...
						_iReadTagRetry:=_iReadTagRetry+1;
					END_IF
				END_IF
				//TEST retry //TEST ONLY
				IF _iReadTagTestRereadN > 0 THEN
					IF _iReadTagTestRereadN > _iReadTagRetry THEN
						_readTagCmd := TRUE;//retry...
						_iReadTagRetry:=_iReadTagRetry+1;
					END_IF
				END_IF
		END_CASE
	ELSE
		_execPulseGenerator(IN := TRUE, PT := T#100MS);	
	END_IF
ELSE
	_iReadTagRetry:= 0;
END_IF
END_METHOD

METHOD SignalClear_ADR_and_RESTART : BOOL
VAR_INPUT
END_VAR
//clear at START and END of reading
IoBisL405Rfid.Restart:= FALSE;
IoBisL405Rfid.Address:= FALSE;
END_METHOD

METHOD SignalGet_ADR : BOOL
VAR_INPUT
END_VAR
//NB: Signals 'Restart' and 'Address' are inverted!
SignalGet_ADR:= IoBisL405Rfid.Restart;
END_METHOD

METHOD SignalGet_RESTART : BOOL
VAR_INPUT
END_VAR
//NB: Signals 'Restart' and 'Address' are inverted!
SignalGet_RESTART:= IoBisL405Rfid.Address;
END_METHOD

METHOD SignalSet_ADR : BOOL
VAR_INPUT
	bADRIn : BOOL;
END_VAR
//NB: Signals 'Restart' and 'Address' are inverted!
IoBisL405Rfid.Restart:= bADRIn;
END_METHOD

METHOD SignalSet_RESTART : BOOL
VAR_INPUT
	bRESTARTIn : BOOL;
END_VAR
//NB: Signals 'Restart' and 'Address' are inverted!
IoBisL405Rfid.Address:= bRESTARTIn;
END_METHOD

METHOD SignalsGet_DataByte : BYTE
VAR_INPUT
END_VAR
SignalsGet_DataByte :=	BOOL_TO_BYTE(IoBisL405Rfid.DataOutput0) +
						(BOOL_TO_BYTE(IoBisL405Rfid.DataOutput1) * 2) +
						(BOOL_TO_BYTE(IoBisL405Rfid.DataOutput2) * 4) +
						(BOOL_TO_BYTE(IoBisL405Rfid.DataOutput3) * 8) +
						(BOOL_TO_BYTE(IoBisL405Rfid.DataOutput4) * 16) +
						(BOOL_TO_BYTE(IoBisL405Rfid.DataOutput5) * 32) +
						(BOOL_TO_BYTE(IoBisL405Rfid.DataOutput6) * 64) +
						(BOOL_TO_BYTE(IoBisL405Rfid.DataOutput7) * 128);
END_METHOD

METHOD Toggle_ADR : BOOL
VAR_INPUT
END_VAR
Toggle_ADR:= FALSE;
IF _iToggleAddress = 1 THEN
	Toggle_ADR:= TRUE;
	IF _bLatchStrobeChanged THEN //only toggle 'ADR' AFTER STR signal change recieved
		_bLatchStrobeChanged:= FALSE; //Clear
		_bLatchADRToggled:=TRUE; //EC//20240710 AAA Smells redundant
		IF SignalGet_ADR() THEN
			SignalSet_ADR(FALSE);
		ELSE
			SignalSet_ADR(TRUE);
		END_IF
		_iToggleAddress:= 1;//(continue toggling)
	END_IF
END_IF
END_METHOD

METHOD Toggle_RESTART : BOOL
VAR_INPUT
END_VAR
Toggle_RESTART:= FALSE;
IF _iDoReset = 1 THEN
	Toggle_RESTART:= TRUE;
	IF SignalGet_RESTART() THEN
		SignalSet_RESTART(FALSE);
		_iDoReset:= 0; //DONE
		_iToggleAddress:= 1;//after restart, ask for data bits
	ELSE
		SignalSet_RESTART(TRUE);
	END_IF
END_IF
END_METHOD

END_FUNCTION_BLOCK

// ---- PMShared/Hardware/Devices/Rfids/RfidBase.TcPOU
FUNCTION_BLOCK ABSTRACT RfidBase EXTENDS TExecution IMPLEMENTS IDevice
VAR_INPUT
END_VAR
VAR_OUTPUT
END_VAR
VAR
	{attribute 'OPC.UA.DA' := '0'}
	_name : STRING;
	{attribute 'OPC.UA.DA' := '0'}
	_deviceID : STRING;				
	{attribute 'OPC.UA.DA' := '0'}	
	_family : DeviceFamily;	
	{attribute 'OPC.UA.DA' := '0'}
	_logger : Logger;
	{attribute 'OPC.UA.DA' := '0'}
	_message : StringBuilder;
	{attribute 'OPC.UA.DA' := '0'}
	_rfidConfig : DeviceConfiguration;	
END_VAR

PROPERTY DeviceID : STRING
GET
DeviceID := _deviceID;
END_GET
SET
_deviceID := DeviceID;
END_SET
END_PROPERTY

PROPERTY Family : DeviceFamily
GET
Family := _family;
END_GET
SET
_family := Family;
END_SET
END_PROPERTY

PROPERTY Name : STRING
GET
Name := _name;
END_GET
SET
_name := Name;
END_SET
END_PROPERTY

END_FUNCTION_BLOCK

// ---- Service/PMs/Psd/Communication/RS232/PsdBkgrdSerialCom.TcPOU
PROGRAM PsdBkgrdSerialCom
VAR_INPUT
	Config : PsdConfig;
END_VAR
VAR
END_VAR

// ScreensConfigs
IF Config.ScreenConfigs.DM430GNScreenConfigFS.IsEnabled THEN
	BkgrdSerialScreenFS();
END_IF
IF Config.ScreenConfigs.DM430GNScreenConfigBS.IsEnabled THEN
	BkgrdSerialScreenBS();
END_IF

END_PROGRAM

// ---- PMShared/Hardware/Devices/Screens/Configs/SerialCommunication/BkgrdSerialScreenFS.TcPOU
PROGRAM BkgrdSerialScreenFS
VAR
	(* background communication with the EL6002 terminal *)
	serialLineCtrl		: SerialLineControl;
	serialLineCtrlError	: BOOL;
	serialLineCtrlErrorID : ComError_t;
	(* 	I/O variables for a EL6002 terminal*)
	stInScreenFS  AT %I*	: EL6inData22B;	
	stOutScreenFS AT %Q*	: EL6outData22B;
END_VAR

(*
The SerialLineControl function block is supposed to be called in every PLC cycle.
It communicates with the serial line hardware device and transmits or receives data.
The SerialLineControl can be called in the standard task (e.g.for PcCOM port usage) 
or in a separate fast task (e.g.for terminal usage) as well.
A fast separate task will be necessary at high baud rates or with KL6001 terminals 
which have a small process image (3 or 5 data bytes only)
*)

(* background communication with the EL6002 terminal *)
serialLineCtrl(
	Mode:= SERIALLINEMODE_EL6_22B, 
	pComIn:= ADR(stInScreenFS), 
	pComOut:= ADR(stOutScreenFS), 
	SizeComIn:= SIZEOF(stInScreenFS), 
	TxBuffer:= HardwareGlobalVariables.TxBufferDM430GNScreenFS, 
	RxBuffer:= HardwareGlobalVariables.RxBufferDM430GNScreenFS
);

IF serialLineCtrl.Error THEN
	serialLineCtrlError := TRUE;
	serialLineCtrlErrorID := serialLineCtrl.ErrorID;
END_IF

END_PROGRAM

// ---- PMShared/Hardware/Devices/Screens/Configs/SerialCommunication/BkgrdSerialScreenBS.TcPOU
PROGRAM BkgrdSerialScreenBS
VAR
	(* background communication with the EL6002 terminal *)
	serialLineCtrl		: SerialLineControl;
	serialLineCtrlError	: BOOL;
	serialLineCtrlErrorID : ComError_t;
	(* 	I/O variables for a EL6002 terminal*)
	stInScreenBS  AT %I*	: EL6inData22B;	
	stOutScreenBS AT %Q*	: EL6outData22B;
END_VAR

(*
The SerialLineControl function block is supposed to be called in every PLC cycle.
It communicates with the serial line hardware device and transmits or receives data.
The SerialLineControl can be called in the standard task (e.g.for PcCOM port usage) 
or in a separate fast task (e.g.for terminal usage) as well.
A fast separate task will be necessary at high baud rates or with KL6001 terminals 
which have a small process image (3 or 5 data bytes only)
*)

(* background communication with the EL6002 terminal *)
serialLineCtrl(
	Mode:= SERIALLINEMODE_EL6_22B, 
	pComIn:= ADR(stInScreenBS), 
	pComOut:= ADR(stOutScreenBS), 
	SizeComIn:= SIZEOF(stInScreenBS), 
	TxBuffer:= HardwareGlobalVariables.TxBufferDM430GNScreenBS, 
	RxBuffer:= HardwareGlobalVariables.RxBufferDM430GNScreenBS
);

IF serialLineCtrl.Error THEN
	serialLineCtrlError := TRUE;
	serialLineCtrlErrorID := serialLineCtrl.ErrorID;
END_IF

END_PROGRAM

// ---- Service/PMs/Nst/Nst.TcPOU
FUNCTION_BLOCK Nst EXTENDS PlcModule
VAR_INPUT
	
	{attribute 'OPC.UA.DA' := '0'}
	NstConfig : NstConfig;
		
	(* AttenuationFilterConfigs *) 
	FW212CAttenuationFilter : FW212CAttenuationFilter(Config := NstConfig.AttenuationFilterConfigs.FW212CAttenuationFilterConfig);
	ELL14KAttenuationFilter : ELL14KAttenuationFilter(Config := NstConfig.AttenuationFilterConfigs.ELL14kAttenuationFilterConfig);
	ELL9AttenuationFilter : ELL9AttenuationFilter(Config := NstConfig.AttenuationFilterConfigs.ELL9AttenuationFilterConfig);
	
	(* LaserConfigs *) 
	SMD12Laser : SMD12Laser(Config := NstConfig.LaserConfigs.SMD12LaserConfig);
	Piano450Laser : Piano450Laser(Config := NstConfig.LaserConfigs.Piano450LaserConfig);
	
	(* ShutterConfigs *)
	Ed12dssShutter : Ed12dssShutter(Config := NstConfig.ShutterConfigs.Ed12dssShutterConfig);
	Sh10pilShutter : Sh10pilShutter(Config := NstConfig.ShutterConfigs.Sh10pilShutterConfig);
	
	(* FastAttenuationConfigs *)
	Std900FastAttenuation : Std900FastAttenuation(Config := NstConfig.FastAttenuationConfigs.Std900FastAttenuationConfig);
	
	(* Ffu *)
	Ffu : Astrofan612Ffu(Config := NstConfig.FfuConfigs.Astrofan612FfuConfig);

	
	(* IonizerConfigs *)
	SJH108Ionizer : SJH108Ionizer(Config := NstConfig.IonizerConfigs.SJH108IonizerConfig);
	
	SmokeDetectedMsg : STRING(255);
	SmokeDetectorFaultMsg : STRING(255);
	VacuumDetectorMsg : STRING(255);
	
	{attribute 'OPC.UA.DA' := '0'}
	_deliverMessages : INT;
	
	{attribute 'OPC.UA.DA' := '0'}
	_execStartTrigger : BOOL;
	{attribute 'OPC.UA.DA' := '0'}
	_execSmokeDetectorResetAlarm : BOOL;
	
	{attribute 'OPC.UA.DA' := '0'}
	_stateTrigCmd : INT;
	{attribute 'OPC.UA.DA' := '0'}
	_stateSmokeCmd : INT;
	{attribute 'OPC.UA.DA' := '0'}
	_stateSmokeResetAlarmCmd : INT;
	{attribute 'OPC.UA.DA' := '0'}
	_setPeriod_ms : LREAL := 100;
	
	{attribute 'OPC.UA.DA' := '0'}
	timerDelayOn : LTON;
	{attribute 'OPC.UA.DA' := '0'}
	timerDelayOff: LTON;	
	{attribute 'OPC.UA.DA' := '0'}
	pulseFlag : BOOL;
	{attribute 'OPC.UA.DA' := '0'}	
	trigOff : BOOL;	
	{attribute 'OPC.UA.DA' := '0'}
	OutputTriggerPlc	AT %Q* : BOOL;
		
	{attribute 'OPC.UA.DA' := '0'}
	InputSmokeDetector_NoFault AT %I* : BOOL;
	{attribute 'OPC.UA.DA' := '0'}
	InputSmokeDetector_Fault AT %I* : BOOL;
	{attribute 'OPC.UA.DA' := '0'}
	InputSmokeDetector_Fire1 AT %I* : BOOL;
	{attribute 'OPC.UA.DA' := '0'}
	InputSmokeDetector_Action AT %I* : BOOL;
	{attribute 'OPC.UA.DA' := '0'}
	InputVacuumIsReady AT %I* : BOOL;
	{attribute 'OPC.UA.DA' := '0'}
	OutputSmokeDetector_ResetAlarm AT %Q* : BOOL;
		
	{attribute 'OPC.UA.DA' := '0'}
	risingEdge : R_TRIG;
	{attribute 'OPC.UA.DA' := '0'}
	_pulseGenerator : TON;	
	{attribute 'OPC.UA.DA' := '0'}
	pulseGeneratorSmokeDetector : TP;
	{attribute 'OPC.UA.DA' := '0'}
	waitSmokeDetected : TP;
	{attribute 'OPC.UA.DA' := '0'}
	smokeDetected : BOOL;	
	{attribute 'OPC.UA.DA' := '0'}
	elapsedTime : STRING;	
	
	{attribute 'OPC.UA.DA' := '0'}
	sensorDetectorFault : BOOL;	
END_VAR
VAR_OUTPUT
END_VAR
VAR			
END_VAR

SUPER^();

(* Attenuation *)
IF NstConfig.AttenuationFilterConfigs.FW212CAttenuationFilterConfig.IsEnabled THEN		
	FW212CAttenuationFilter();
	IF FW212CAttenuationFilter.InitConfigSerialCom THEN
		;
	END_IF
ELSIF NstConfig.AttenuationFilterConfigs.ELL14KAttenuationFilterConfig.IsEnabled THEN		
	ELL14KAttenuationFilter();
	IF ELL14KAttenuationFilter.InitConfigSerialCom THEN
		;
	END_IF	
ELSIF NstConfig.AttenuationFilterConfigs.ELL9AttenuationFilterConfig.IsEnabled THEN		
	ELL9AttenuationFilter();
	IF ELL9AttenuationFilter.InitConfigSerialCom THEN
		;
	END_IF	
END_IF

(* Laser *)
IF NstConfig.LaserConfigs.SMD12LaserConfig.IsEnabled THEN
	SMD12Laser();
	IF SMD12Laser.InitConfigSerialCom THEN
		;
	END_IF
ELSIF NstConfig.LaserConfigs.Piano450LaserConfig.IsEnabled THEN
	Piano450Laser();
	IF Piano450Laser.InitConfigSerialCom THEN
		;
	END_IF
END_IF

(* Shutter *)
IF NstConfig.ShutterConfigs.Ed12dssShutterConfig.IsEnabled THEN
	Ed12dssShutter();	
ELSIF NstConfig.ShutterConfigs.SH10PILShutterConfig.IsEnabled THEN
	Sh10pilShutter();
END_IF

(* Fast attenuation *)
IF NstConfig.FastAttenuationConfigs.Std900FastAttenuationConfig.IsEnabled THEN
	Std900FastAttenuation();	
END_IF

(*FFU*)
IF NstConfig.FfuConfigs.Astrofan612FfuConfig.IsEnabled THEN
	Ffu();
END_IF

(* Ionizer *)
IF NstConfig.IonizerConfigs.SJH108IonizerConfig.IsEnabled THEN
	SJH108Ionizer();
END_IF

TriggerOutEmitSignal(_execStartTrigger, _setPeriod_ms);
SmokeDetectorResetAlarm(_execSmokeDetectorResetAlarm);

CASE _deliverMessages OF
	EFeedbackMsgPlc.SmokeDetectedMsg:
		SmokeDetectedMsg := message;
	EFeedbackMsgPlc.SmokeDetectorFaultMsg:
		SmokeDetectorFaultMsg := message;			
	EFeedbackMsgPlc.VacuumDetectorMsg:
		VacuumDetectorMsg := message;
END_CASE

IF (NOT _execStartTrigger) THEN
	MessageScheduler();
END_IF

METHOD FB_init : BOOL
VAR_INPUT
	bInitRetains : BOOL; // if TRUE, the retain variables are initialized (warm start / cold start)
	bInCopyCode : BOOL;  // if TRUE, the instance afterwards gets moved into the copy code (online change)
	Config : NstConfig;
END_VAR
NstConfig := Config;
NstBkgrdLsSerialCom(Config := NstConfig);

IF Config.IsEnabled THEN
	_logger.Information('NST devices initialization starting...');
END_IF	

(* AttenuationFilterConfigs *)
IF Config.AttenuationFilterConfigs.FW212CAttenuationFilterConfig.IsEnabled THEN
	FW212CAttenuationFilter.FB_init(FALSE, FALSE, Config := Config.AttenuationFilterConfigs.FW212CAttenuationFilterConfig);	
ELSIF Config.AttenuationFilterConfigs.ELL14kAttenuationFilterConfig.IsEnabled THEN
	ELL14KAttenuationFilter.FB_init(FALSE, FALSE, Config := Config.AttenuationFilterConfigs.ELL14kAttenuationFilterConfig);
ELSIF Config.AttenuationFilterConfigs.ELL9AttenuationFilterConfig.IsEnabled THEN
	ELL9AttenuationFilter.FB_init(FALSE, FALSE, Config := Config.AttenuationFilterConfigs.ELL9AttenuationFilterConfig);	
END_IF

(* LaserConfigs *) 
IF Config.LaserConfigs.SMD12LaserConfig.IsEnabled THEN
	SMD12Laser.FB_init(FALSE, FALSE, Config := Config.LaserConfigs.SMD12LaserConfig);
ELSIF Config.LaserConfigs.Piano450LaserConfig.IsEnabled THEN
	Piano450Laser.FB_init(FALSE, FALSE, Config := Config.LaserConfigs.Piano450LaserConfig);	
END_IF

(* ShutterConfigs *) 
IF Config.ShutterConfigs.Ed12dssShutterConfig.IsEnabled THEN
	Ed12dssShutter.FB_init(FALSE, FALSE, Config := Config.ShutterConfigs.Ed12dssShutterConfig);	
ELSIF Config.ShutterConfigs.Sh10pilShutterConfig.IsEnabled THEN
	Sh10pilShutter.FB_init(FALSE, FALSE, Config := Config.ShutterConfigs.Sh10pilShutterConfig);		
END_IF

(* FastAttenuationConigs *)
IF Config.FastAttenuationConfigs.Std900FastAttenuationConfig.IsEnabled THEN
	Std900FastAttenuation.FB_init(FALSE, FALSE, Config := Config.FastAttenuationConfigs.Std900FastAttenuationConfig);	
END_IF

(* IonizerConfig *)
IF Config.IonizerConfigs.SJH108IonizerConfig.IsEnabled THEN
	SJH108Ionizer.FB_init(FALSE, FALSE, Config := Config.IonizerConfigs.SJH108IonizerConfig);	
END_IF

(* Ffu *) 
IF Config.FfuConfigs.Astrofan612FfuConfig.IsEnabled THEN
	Ffu.FB_init(FALSE, FALSE, Config := Config.FfuConfigs.Astrofan612FfuConfig);	
END_IF

IF Config.IsEnabled THEN
	_logger.Information('NST devices initialization ended...');
END_IF
END_METHOD

METHOD MessageScheduler
VAR_INPUT
END_VAR
IF _pulseGenerator.Q THEN
	_pulseGenerator(IN := FALSE, PT := T#10MS);
		
	CASE _itemScheduler OF		
		0:	SmokeDetector();
			_itemScheduler := 1;
			
		1: VacuumDetector();
			_itemScheduler := 0;
	END_CASE
ELSE
	_pulseGenerator(IN := TRUE, PT := T#1S);		
END_IF
END_METHOD

METHOD PROTECTED SmokeDetector 
VAR
	engagesEMO : INT := 10;
END_VAR
_deliverMessages := EFeedbackMsgPlc.SmokeDetectedMsg;

IF InputSmokeDetector_Fire1 OR InputSmokeDetector_Action THEN
	CASE _stateSmokeCmd OF	
		0: _logger.Information(_message.Reset().
								Append('Smoke detected').ToString());
			smokeDetected := TRUE;
			_stateSmokeCmd := 1;
	END_CASE
END_IF

IF _stateSmokeCmd = 1 THEN		
	waitSmokeDetected(IN := smokeDetected, PT := T#30S);			
	IF waitSmokeDetected.Q THEN
		IF OutputSmokeDetector_ResetAlarm THEN
			IF smokeDetected THEN
				_logger.Information(_message.Reset().Append('Stop smoke detected').ToString());	
			END_IF									
			smokeDetected := FALSE;	
		END_IF
	ELSE
		IF smokeDetected AND _stateSmokeCmd <> engagesEMO THEN	
			_logger.Warning(_message.Reset().Append('Time limit has expired. Safety PLC must restart machine').ToString());			
		END_IF		
		_stateSmokeCmd := engagesEMO;
	END_IF												
	
	// Reset waitSmokeDetected
	IF NOT smokeDetected AND NOT waitSmokeDetected.Q THEN
		_stateSmokeCmd := 0;
		InputSmokeDetector_Fire1 := FALSE;
		InputSmokeDetector_Action := FALSE;
	END_IF
	
ELSE
	smokeDetected := FALSE;
END_IF

IF _stateSmokeCmd <> engagesEMO THEN	
	message := BOOL_TO_STRING(smokeDetected);	
END_IF
END_METHOD

METHOD PROTECTED SmokeDetectorFault
VAR_INPUT
END_VAR
_deliverMessages := EFeedbackMsgPlc.SmokeDetectorFaultMsg;

IF InputSmokeDetector_Fault THEN
	sensorDetectorFault := TRUE;
ELSE
	sensorDetectorFault := FALSE;
END_IF

IF sensorDetectorFault THEN
	sensorDetectorFault := FALSE;
	message := 'Fault'; 	
END_IF
END_METHOD

{attribute 'TcRpcEnable' := '1'}
METHOD PROTECTED SmokeDetectorResetAlarm : BOOL;
VAR_INPUT
	Execute : BOOL;
END_VAR
VAR
	{attribute 'OPC.UA.DA' := '0'}
	smokeDetectorResetAlarmTrig : BOOL;
END_VAR
IF Execute THEN
	_execSmokeDetectorResetAlarm := TRUE;

	CASE _stateSmokeResetAlarmCmd OF	
		0:  _logger.Information(_message.Reset().
								Append('Smoke detector alarm reset triggered').ToString());
			
			smokeDetectorResetAlarmTrig := TRUE;
			_stateSmokeResetAlarmCmd := 1;	 
	END_CASE
			
	pulseGeneratorSmokeDetector(In := smokeDetectorResetAlarmTrig, PT := T#3S);					
	smokeDetectorResetAlarmTrig := pulseGeneratorSmokeDetector.Q; 	
	
	IF NOT pulseGeneratorSmokeDetector.Q AND pulseGeneratorSmokeDetector.ET = T#0S THEN		
		OutputSmokeDetector_ResetAlarm := FALSE;
		
		_execSmokeDetectorResetAlarm := FALSE;
		_stateSmokeResetAlarmCmd := 0;
	END_IF						
	
	OutputSmokeDetector_ResetAlarm := smokeDetectorResetAlarmTrig;
	SmokeDetectorResetAlarm := smokeDetectorResetAlarmTrig;
END_IF
END_METHOD

{attribute 'TcRpcEnable' := '1'}
METHOD PROTECTED TriggerOutEmitSignal
VAR_INPUT
	Execute : BOOL;
	PulseDuration_ms : LREAL;	
END_VAR
VAR
	duration_ms : LTIME;
END_VAR

IF Execute THEN
	_execStartTrigger := TRUE;
	_setPeriod_ms := PulseDuration_ms;
	
	CASE _stateTrigCmd OF		
		0:	OutputTriggerPlc := _execStartTrigger AND NOT trigOff;	
			_stateTrigCmd := 1;	
					
		1:	IF trigOff = TRUE THEN
				OutputTriggerPlc := FALSE;
				_stateTrigCmd := 2;						
			END_IF
			
			timerDelayOff(IN := OutputTriggerPlc, PT := LREAL_TO_LTIME(_setPeriod_ms * 1E+6));
			trigOff := timerDelayOff.Q;	
								
		2:	_execStartTrigger := FALSE;	
			_stateTrigCmd := 0;
	END_CASE
END_IF
END_METHOD

METHOD VacuumDetector : BOOL
VAR_INPUT
END_VAR
_deliverMessages := EFeedbackMsgPlc.VacuumDetectorMsg;

IF InputVacuumIsReady THEN
	VacuumDetector := TRUE;
ELSE
	VacuumDetector := FALSE;
END_IF

message := BOOL_TO_STRING(VacuumDetector);
END_METHOD

END_FUNCTION_BLOCK

// ---- PMShared/Hardware/Devices/Lasers/Leukos/Piano450Laser.TcPOU
{attribute 'OPC.UA.DA' := '1'}
FUNCTION_BLOCK Piano450Laser EXTENDS LaserBase
VAR_INPUT
END_VAR
VAR_OUTPUT
END_VAR
VAR
	{attribute 'OPC.UA.DA' := '0'}
	_config : Piano450LaserConfig;	
	{attribute 'OPC.UA.DA' := '0'}
	_coeAccess : CoeAccess;	
	{attribute 'OPC.UA.DA' := '0'}
	_initConfigSerialCom : BOOL;	
	{attribute 'OPC.UA.DA' := '0'}
	sReplyPrefix4 : STRING(4) := '>'; //DEFINE expected device reply string start sequence
	{attribute 'OPC.UA.DA' := '0'}
	iReplyPrefixLen : INT := LEN(sReplyPrefix4);
	{attribute 'OPC.UA.DA' := '0'}
	sReplySuffix4 : STRING(4) := Const.LF_CR; //DEFINE expected device reply string termination sequence
	{attribute 'OPC.UA.DA' := '0'}
	iReplySuffixLen : INT := LEN(sReplySuffix4);
	{attribute 'OPC.UA.DA' := '0'}
	_serialCom  : SerialCom(Prefix :='', Suffix := sReplySuffix4);
	{attribute 'OPC.UA.DA' := '0'}
	_refSerialCom : REFERENCE TO SerialCom(Prefix :='', Suffix := sReplySuffix4) := _serialCom;		 
	{attribute 'OPC.UA.DA' := '0'}
	_isReceived : BOOL;
	
	{attribute 'OPC.UA.DA' := '0'}
	_deliverMessages : INT;
		
	StateMsg : STRING(255);
	StatusMsg : STRING(255);
	IsAliveMsg : STRING(255);
	PowerMsg : STRING(255);
	InterlockStatusMsg : STRING(255);
	LaserTemperatureMsg : STRING(255);
	CrystalTemperatureMsg : STRING(255);
	RunningTimeLaserOnMsg : STRING(255);
	RunningTimeElectroOnMsg : STRING(255);		
	CustomMsg : STRING(255);	
	
	{attribute 'OPC.UA.DA' := '0'}
	crystalTemp : REAL;
	{attribute 'OPC.UA.DA' := '0'} 
	laserTemp : REAL;
	{attribute 'OPC.UA.DA' := '0'} 
	interlockTemp : STRING;
		
	{region 'Commands'}
	
	{attribute 'OPC.UA.DA' := '0'}
	_powerOn : BOOL;
	{attribute 'OPC.UA.DA' := '0'}
	_powerOff : BOOL;
	{attribute 'OPC.UA.DA' := '0'}
	_setPowerCmd : BOOL;
	{attribute 'OPC.UA.DA' := '0'}	 
	_setCurrentCmd : BOOL;
	{attribute 'OPC.UA.DA' := '0'}			 
	_controlModeCmd : BOOL;
	{attribute 'OPC.UA.DA' := '0'}
	_customCmd : BOOL;	
	{attribute 'OPC.UA.DA' := '0'}			  		   
	_raiseProperties : BOOL;
	
	{endregion}			
	
	{attribute 'OPC.UA.DA' := '0'}
	_initDevice : BOOL;	
	 
	{attribute 'OPC.UA.DA' := '0'}
	_cmd : STRING;			
	{attribute 'OPC.UA.DA' := '0'}
	_setpoint : LREAL := 0;
	{attribute 'OPC.UA.DA' := '0'}
	_itemScheduler : INT;
	{attribute 'OPC.UA.DA' := '0'}
	_itemExecScheduler : INT;		
	{attribute 'OPC.UA.DA' := '0'}
	_itemRaisedProperties : INT;			
	{attribute 'OPC.UA.DA' := '0'}
	_pulseGenerator : TON;	
	{attribute 'OPC.UA.DA' := '0'}
	_execPulseGenerator : TON;	
	{attribute 'OPC.UA.DA' := '0'}
	_pulseIsAliveGenerator : TON;	
	
	{attribute 'OPC.UA.DA' := '0'}
	message : STRING;
	{attribute 'OPC.UA.DA' := '0'}	
	_length : INT;
	{attribute 'OPC.UA.DA' := '0'}
	sSubStr4 : STRING(4) := '';
	{attribute 'OPC.UA.DA' := '0'}
	_mode : EControlModeSmd12;	
	
	{attribute 'OPC.UA.DA' := '0'}
	_lifeTimeCount : UINT;
	{attribute 'OPC.UA.DA' := '0'}
	_notifyIsAlive : BOOL;
	
END_VAR

IF NOT InitConfigSerialCom THEN
	ConfigureSerialCom();
ELSIF THIS^.Status = TExecutionState.Ready THEN
	IF _refSerialCom.ErrorReceiveId = COMERROR_NOERROR THEN
		_refSerialCom(TxBuffer:= HardwareGlobalVariables.TxBufferLaser, 
		 	      	  RxBuffer:= HardwareGlobalVariables.RxBufferLaser);
	END_IF				  
	
	// Init device
	InitDevice(); 				  				 

	// Check if it's still alive	
	IF _notifyIsAlive THEN
		IsAliveMsg := TO_STRING(_lifeTimeCount);
		_notifyIsAlive := FALSE;
	END_IF		
	
	// Deliver messages
	IF _refSerialCom.IsReceived THEN				 	
		CASE _deliverMessages OF			
			EFeedbackMsgPiano450.StatusMsg :
			_length := LEN(_refSerialCom.LastReceivedString);	
				IF _length = 4 THEN
					sSubStr4 := RIGHT(_refSerialCom.LastReceivedString, iReplySuffixLen);
					IF sSubStr4 = sReplySuffix4 THEN
						sSubStr4 := LEFT(_refSerialCom.LastReceivedString, iReplyPrefixLen);
						IF sSubStr4 = sReplyPrefix4 THEN
							StatusMsg := LEFT(_refSerialCom.LastReceivedString, 2);
							StatusMsg := DELETE(StatusMsg, 1, 1);//remove 1st character
						END_IF
					END_IF
				END_IF		
								
			EFeedbackMsgPiano450.InterlockStatusMsg :
			_length := LEN(_refSerialCom.LastReceivedString);	
				IF _length = 9 THEN
					sSubStr4 := RIGHT(_refSerialCom.LastReceivedString, iReplySuffixLen);
					IF sSubStr4 = sReplySuffix4 THEN
						sSubStr4 := LEFT(_refSerialCom.LastReceivedString, iReplyPrefixLen);
						IF sSubStr4 = sReplyPrefix4 THEN
							InterlockStatusMsg := LEFT(_refSerialCom.LastReceivedString, 7);													
							interlockTemp := CONCAT('2#', DELETE(InterlockStatusMsg, 1, 1));
							
							InterlockStatusMsg := TranslateStatusLaser(STRING_TO_BYTE(interlockTemp));
						END_IF
					END_IF
				END_IF
				
			EFeedbackMsgPiano450.LaserTemperatureMsg :
				_length := LEN(_refSerialCom.LastReceivedString);	
				IF _length = 11 THEN
					sSubStr4 := RIGHT(_refSerialCom.LastReceivedString, iReplySuffixLen);
					IF sSubStr4 = sReplySuffix4 THEN
						sSubStr4 := LEFT(_refSerialCom.LastReceivedString, iReplyPrefixLen);
						IF sSubStr4 = sReplyPrefix4 THEN
							LaserTemperatureMsg := LEFT(_refSerialCom.LastReceivedString, 9);
							LaserTemperatureMsg := DELETE(LaserTemperatureMsg, 1, 1);//remove 1st character
							
							laserTemp := STRING_TO_REAL(DELETE(LaserTemperatureMsg, 4, 1)) + 45; // Add 45 °C
							LaserTemperatureMsg := REAL_TO_STRING(laserTemp);
						END_IF
					END_IF
				END_IF
				
			EFeedbackMsgPiano450.CrystalTemperatureMsg :
				_length := LEN(_refSerialCom.LastReceivedString);	
				IF _length = 11 THEN
					sSubStr4 := RIGHT(_refSerialCom.LastReceivedString, iReplySuffixLen);
					IF sSubStr4 = sReplySuffix4 THEN
						sSubStr4 := LEFT(_refSerialCom.LastReceivedString, iReplyPrefixLen);
						IF sSubStr4 = sReplyPrefix4 THEN
							CrystalTemperatureMsg := LEFT(_refSerialCom.LastReceivedString, 9);
							CrystalTemperatureMsg := DELETE(CrystalTemperatureMsg, 1, 1);//remove 1st character
							
							crystalTemp := STRING_TO_REAL(DELETE(CrystalTemperatureMsg, 4, 4)) * 0.01;							
							CrystalTemperatureMsg:= REAL_TO_STRING(crystalTemp);							
						END_IF
					END_IF
				END_IF
				
			EFeedbackMsgPiano450.CustomMsg :
				CustomMsg := _refSerialCom.LastReceivedString;			
		END_CASE
	ELSE
		CASE _deliverMessages OF			
			EFeedbackMsgPiano450.StateMsg :
				StateMsg := ANY_TO_STRING(State);
		END_CASE
	END_IF								   							   	
	
	PowerOn(_powerOn);
	PowerOff(_powerOff);	
	CustomCommand(_customCmd, _cmd);
	RaisePropertiesChanged(_raiseProperties);
	
	IF (NOT _powerOn AND NOT _powerOff AND NOT _customCmd AND NOT _raiseProperties) THEN
		MessageScheduler();
	END_IF
END_IF

METHOD ConfigureSerialCom
VAR_INPUT
END_VAR
IF _coeAccess.CoeOperation.Ready THEN
	_logger.Information(_message.Reset().Append('Start configuration com serial').ToString());
END_IF;	

_coeAccess.CoeOperation.Start();
_coeAccess(SerialCommunication := _config.SerialCommunication);
	
IF _coeAccess.CoeOperation.Done THEN
	_coeAccess.SetDone();	
	
	_Logger.Information(_message.Reset().
							Append('{').Append(TO_STRING(THIS^.Family)).Append('} : ').
							Append(' - Status : ').Append(TO_STRING(_coeAccess.Status)).ToString());	
	InitConfigSerialCom := TRUE;
END_IF
 
IF _coeAccess.CoeOperation.Error THEN	
	_coeAccess.SetError(0);
	
	_Logger.Error(_message.Reset().
							Append('{').Append(TO_STRING(THIS^.Family)).Append('} : ').
							Append(' - Status : ').Append(TO_STRING(_coeAccess.Status)).ToString());
	InitConfigSerialCom := TRUE;
END_IF

THIS^.Status := _coeAccess.Status;
State := _coeAccess.Status;
END_METHOD

METHOD ControlMode
VAR_INPUT
	Execute : BOOL;
	Mode : EControlModeSmd12;
END_VAR
VAR
//	currentModecmd : STRING := 'CONTROL=CURRENT';
//	powerModecmd : STRING := 'CONTROL=POWER';
END_VAR
IF Execute THEN
//	_logger.Information(_message.Reset().
//								Append(_config.Name).
//								Append(' - ControlMode : ').Append(TO_STRING(Mode)).ToString());
//	
//	IF MODE = EControlModeSmd12.CurrentMode THEN
//		_serialCom.Send(currentModecmd);
//	ELSIF MODE = EControlModeSmd12.PowerMode THEN
//		_serialCom.Send(powerModecmd);
//	END_IF
//	
	_controlModeCmd := FALSE;		
END_IF
END_METHOD

{attribute 'TcRpcEnable' := '1'}
(** Custom command **)
METHOD CustomCommand
VAR_INPUT
	Execute : BOOL;
	Cmd : STRING;
END_VAR
IF Execute THEN
	_logger.Information(_message.Reset().
								Append(_config.Name).
								Append(' - Custom command : ').
								Append(Cmd).ToString());	
	_deliverMessages := EFeedbackMsgSMD12.CustomMsg;														
	_serialCom.Send(Cmd);	
	_customCmd := FALSE;
END_IF
END_METHOD

METHOD FB_init : BOOL
VAR_INPUT
	bInitRetains : BOOL; // if TRUE, the retain variables are initialized (warm start / cold start)
	bInCopyCode : BOOL;  // if TRUE, the instance afterwards gets moved into the copy code (online change)
	Config : Piano450LaserConfig;
END_VAR
IF Config.IsEnabled THEN
	_config := Config;
	
	SUPER^._laserConfig.Name := Config.Name;
	SUPER^._laserConfig.DeviceID := Config.DeviceID;
	SUPER^._laserConfig.IsEnabled := Config.IsEnabled;
	SUPER^._laserConfig.LogLevel := Config.LogLevel;
	
	SUPER^.Name := Config.Name;
	SUPER^.DeviceID := Config.DeviceID;	
	THIS^.Family := DeviceFamily.Laser;
		
	_Logger.Information(_message.Reset().Append('Init ').
							Append('{').Append(TO_STRING(THIS^.Family)).Append('} - ').
							Append('{').Append(TO_STRING(Config.Name)).Append('}').ToString());																													
END_IF
END_METHOD

(** Returns the temperature of the PSU in degrees centigrade **)
METHOD GetCrystalTemperature
VAR_INPUT
END_VAR
VAR
	cmd : STRING := '*mede'; //*mede-> CCCC LLL, CCCC: crystal temperature (0.01 of °C), LLL: laser temperature + 45°C
END_VAR
_deliverMessages := EFeedbackMsgPiano450.CrystalTemperatureMsg;
_serialCom.Send(cmd);
END_METHOD

(** Returns the status of the Interlock **)
METHOD PROTECTED GetInterlockStatus 
VAR_INPUT
END_VAR
VAR
	cmd : STRING := '*regi'; //*regi-> ABCDEE A: Interlock 0:ok 1:nok reboot, B: Laser com 0:ok 1:nok reboot, C: Laser temp 0: Ok 1: nok, D: Peltier 0: Nok 1: Ok, EE: diode 00: Off 01: Computer Off 10: Fully On 11: Modulation On
END_VAR
_deliverMessages := EFeedbackMsgPiano450.InterlockStatusMsg;
_serialCom.Send(cmd);
END_METHOD

(** Return status laser **)
METHOD GetLaserStatus
VAR_INPUT	
END_VAR
VAR
	cmd : STRING := '*lase'; // 0: Laser off - 1: Laser On
END_VAR
_deliverMessages := EFeedbackMsgPiano450.StatusMsg;
_serialCom.Send(cmd);
END_METHOD

(** Returns the temperature of the laser head in degrees centigrade **)
METHOD GetLaserTemperature 
VAR_INPUT
END_VAR
VAR
	cmd : STRING := '*mede'; //*mede-> CCCC LLL, CCCC: crystal temperature (0.01 of °C), LLL: laser temperature + 45°C
END_VAR
_deliverMessages := EFeedbackMsgPiano450.LaserTemperatureMsg;
_serialCom.Send(cmd);
END_METHOD

METHOD GetRunningTimeElectroOnMsg
VAR_INPUT
END_VAR
VAR
	cmd : STRING := '*durl';
END_VAR
_deliverMessages := EFeedbackMsgPiano450.RunningTimeLaserOnMsg;
_serialCom.Send(cmd);
END_METHOD

METHOD GetRunningTimeLaserOnMsg
VAR_INPUT
END_VAR
VAR
	cmd : STRING := '*dura';
END_VAR
_deliverMessages := EFeedbackMsgPiano450.RunningTimeElectroOnMsg;
_serialCom.Send(cmd);
END_METHOD

{attribute 'TcRpcEnable' := '1'}
//*dura-> electronic DDDDdHHhMMmin, DDDD: days, HH: hours, MM: minutes
//*durl-> diode DDDDdHHhMMmin, DDDD: days, HH: hours, MM: minutes
METHOD GetTimers : HoursStruct
VAR_INPUT
	Execute : BOOL;
END_VAR
VAR
	cmd : STRING := '*dura';
END_VAR
IF Execute THEN
	_logger.Information(_message.Reset().
								Append(_config.Name).
								Append(' - GetTimers').ToString());
	_serialCom.Send(cmd);
END_IF
END_METHOD

PROPERTY InitConfigSerialCom : BOOL
GET
InitConfigSerialCom := _initConfigSerialCom;
END_GET
SET
_initConfigSerialCom := InitConfigSerialCom;
END_SET
END_PROPERTY

METHOD InitDevice
VAR_INPUT
END_VAR
IF NOT _initDevice THEN	
	_logger.Information(_message.Reset().
								Append(_config.Name).
								Append(' - InitDevice').ToString());	
	_raiseProperties:= TRUE;	
	_initDevice := TRUE;	
END_IF
END_METHOD

METHOD PROTECTED IsAlive
VAR_INPUT
END_VAR
_notifyIsAlive := TRUE;

IF _lifeTimeCount < 5 THEN
	_lifeTimeCount := _lifeTimeCount + 1;
ELSE
	_lifeTimeCount := 1;
END_IF
END_METHOD

METHOD MessageScheduler
VAR_INPUT
END_VAR
IF _pulseGenerator.Q THEN
	_pulseGenerator(IN := FALSE, PT := T#10MS);
		
	CASE _itemScheduler OF					
		0:	GetLaserStatus(); 
			_itemScheduler := 1;	

		1:	GetInterlockStatus(); 
			_itemScheduler := 2;				
	
		2:  GetLaserTemperature();
			_itemScheduler := 3;	
		
		3:  GetCrystalTemperature();
			_itemScheduler := 0;		
	END_CASE
ELSE
	_pulseGenerator(IN := TRUE, PT := T#100MS);		
END_IF


IF _pulseIsAliveGenerator.Q THEN
	_pulseIsAliveGenerator(IN := FALSE, PT := T#10MS);
		
	IsAlive();	
ELSE
	_pulseIsAliveGenerator(IN := TRUE, PT := T#1000MS);		
END_IF
END_METHOD

{attribute 'TcRpcEnable' := '1'}
(** Disables the laser, regardless of the interlock status **)
METHOD PROTECTED PowerOff
VAR_INPUT
	Execute : BOOL;
END_VAR
VAR
	cmd : STRING := '*lase 0';
END_VAR
IF Execute THEN	
	_powerOff := TRUE;	
	
	IF _execPulseGenerator.Q THEN
		_execPulseGenerator(IN := FALSE, PT := T#10MS);
			
		CASE _itemExecScheduler OF
			0: _logger.Information(_message.Reset().
								Append(_config.Name).
								Append(' - PowerOff').ToString());
				_serialCom.Send(cmd);
				_itemExecScheduler := 1;
			
			1:  GetInterlockStatus();
				_itemExecScheduler := 2;
				
			2:  _powerOff := FALSE;	
				_itemExecScheduler := 0;		
								
		END_CASE
	ELSE
		_execPulseGenerator(IN := TRUE, PT := T#100MS);	
	END_IF
END_IF
END_METHOD

{attribute 'TcRpcEnable' := '1'}
(* Enables the laser subject to Interlock and Enable Switch status *)
METHOD PROTECTED PowerOn
VAR_INPUT
	Execute : BOOL;
END_VAR
VAR
	cmd : STRING := '*lase 1';
END_VAR
IF Execute THEN	
	_powerOn := TRUE;	

	IF _execPulseGenerator.Q THEN
		_execPulseGenerator(IN := FALSE, PT := T#10MS);
			
		CASE _itemExecScheduler OF
			0: _logger.Information(_message.Reset().
								Append(_config.Name).
								Append(' - PowerOn').ToString());
				_serialCom.Send(cmd);
				_itemExecScheduler := 1;
			
			1:  GetInterlockStatus();
				_itemExecScheduler := 2;
				
			2:  _powerOn := FALSE;	
				_itemExecScheduler := 0;		
								
		END_CASE
	ELSE
		_execPulseGenerator(IN := TRUE, PT := T#100MS);	
	END_IF
END_IF
END_METHOD

{attribute 'TcRpcEnable' := '1'}
METHOD RaisePropertiesChanged
VAR_INPUT
	Execute : BOOL;
END_VAR
IF Execute THEN
	_raiseProperties := TRUE;
	
	IF _pulseGenerator.Q THEN
		_pulseGenerator(IN := FALSE, PT := T#10MS);	

		CASE _itemRaisedProperties OF
			0:  StateMsg := ' ';
				StatusMsg := ' ';
			    InterlockStatusMsg := ' ';
				LaserTemperatureMsg := ' ';
				CrystalTemperatureMsg := ' ';
				RunningTimeLaserOnMsg := ' ';
				RunningTimeElectroOnMsg := ' ';
				CustomMsg := ' ';
				
				_itemRaisedProperties := 10;											
			
			10 : GetLaserStatus();
				 _itemRaisedProperties := 11;
				 
			11 : GetInterlockStatus();
				 _itemRaisedProperties := 12;
				 
			12 : GetLaserTemperature();
				 _itemRaisedProperties := 13;
				 
			13 : GetCrystalTemperature();
				 _itemRaisedProperties := 14;
				
			14 : _deliverMessages := EFeedbackMsgPiano450.StateMsg;
				_itemRaisedProperties := 15;
				
			15:  GetRunningTimeLaserOnMsg();
				_itemRaisedProperties := 16;
				
			16:  GetRunningTimeElectroOnMsg();
				_itemRaisedProperties := 17;
				
			17:  _logger.Information(_message.Reset().
								Append(_config.Name).
								Append(' - RaisePropertiesChanged').ToString());
				_raiseProperties := FALSE;				
				_itemRaisedProperties := 0;
			
		END_CASE
	ELSE
		_pulseGenerator(IN := TRUE, PT := T#100MS);	
	END_IF
END_IF
END_METHOD

(** Returns the power of the laser **)
METHOD PROTECTED ReadPower 
VAR_INPUT
END_VAR
VAR
//	cmd : STRING := 'POWER?';
END_VAR
//EC::not available on this device...

//_deliverMessages := EFeedbackMsgSMD12.PowerMsg;
//_serialCom.Send(cmd);
END_METHOD

{attribute 'TcRpcEnable' := '1'}
(** This sets the output power of the laser 
For example, to set a power of 2800 mW, send the string POWER=2800, followed by striking the RETURN key
**)
METHOD PROTECTED SetPower 
VAR_INPUT
	Execute : BOOL;
	Power : LREAL;
END_VAR
VAR
	cmd : STRING := 'POWER=';
END_VAR
//EC//NOT USED on this device!...
IF Execute THEN	
	_setPowerCmd := TRUE;	

	_setpoint := Power;
	
	IF _execPulseGenerator.Q THEN
		_execPulseGenerator(IN := FALSE, PT := T#10MS);
			
		CASE _itemExecScheduler OF
			0: _logger.Information(_message.Reset().
								Append(_config.Name).
								Append(' - SetPower : ').Append(TO_STRING(_setpoint)).ToString());
				_serialCom.Send(CONCAT(cmd, TO_STRING(_setpoint)));
				_itemExecScheduler := 1;
			
			1:  ReadPower();
				_itemExecScheduler := 2;
				
			2:  _setPowerCmd := FALSE;	
				_itemExecScheduler := 0;		
								
		END_CASE
	ELSE
		_execPulseGenerator(IN := TRUE, PT := T#100MS);	
	END_IF
END_IF
END_METHOD

(** he full status of the laser system **)
METHOD TranslateStatusLaser : STRING
VAR_INPUT
	status : BYTE; // Data 	ABCDEE	
END_VAR
VAR
END_VAR

IF (status AND STRING_TO_BYTE('2#100000')) = STRING_TO_BYTE('2#100000') THEN
	// A: Interlock -> 0: no problem - 1: problem interlock (reboot needed)
	TranslateStatusLaser := 'Problem interlock (reboot needed)';
	
ELSIF (status AND STRING_TO_BYTE('2#010000')) = STRING_TO_BYTE('2#010000')  THEN
	// B: Laser head communication -> 0: no problem - 1: problem (reboot needed)
	TranslateStatusLaser := 'Problem (reboot needed)';
	
ELSIF (status AND STRING_TO_BYTE('2#001000')) = STRING_TO_BYTE('2#001000')  THEN
	// C: Laser temperature -> 0: OK - 1:outside the running range
	TranslateStatusLaser := 'Outside the running range';
	
ELSIF (status AND STRING_TO_BYTE('2#000100')) <> STRING_TO_BYTE('2#000100')  THEN
	// D: Peltier regulation status -> 0: Laser non thermalized - 1: Temperature Ok
	TranslateStatusLaser := 'Laser non thermalized';
	
ELSIF (status AND STRING_TO_BYTE('2#000001')) = STRING_TO_BYTE('2#000001') THEN	
	// EE: Status of laser diode -> 00: Off - 01: Computer Off - 10: Fully On - 11: Modulation On	
	TranslateStatusLaser := 'Laser diode - Computer Off';
	
ELSIF (status AND STRING_TO_BYTE('2#000010')) = STRING_TO_BYTE('2#000010') THEN
	// EE: Status of laser diode -> 00: Off - 01: Computer Off - 10: Fully On - 11: Modulation On
	TranslateStatusLaser := 'Laser diode - Fully On';
		
ELSIF (status AND STRING_TO_BYTE('2#000011')) = STRING_TO_BYTE('2#000011') THEN
	// EE: Status of laser diode -> 00: Off - 01: Computer Off - 10: Fully On - 11: Modulation On
	
	TranslateStatusLaser := 'Laser diode - Modulation On';
ELSE
	TranslateStatusLaser := 'OK';	
END_IF
END_METHOD

END_FUNCTION_BLOCK

// ---- PMShared/Hardware/Devices/Ionizers/Keyence/SJH108Ionizer.TcPOU
 {attribute 'OPC.UA.DA' := '1'}
FUNCTION_BLOCK SJH108Ionizer EXTENDS IonizerBase
VAR_INPUT
	
END_VAR
VAR_OUTPUT
END_VAR
VAR
	{attribute 'OPC.UA.DA' := '0'}
	_config : SJH108IonizerConfig;	
	{attribute 'OPC.UA.DA' := '0'}
	IoSJH108A : IoSJH108A;
	
	{attribute 'OPC.UA.DA' := '0'}
	_initDevice : BOOL;	
	
	{region 'Commands'}	
		 	
	{attribute 'OPC.UA.DA' := '0'}
	_openAirValveCmd : BOOL;	
	{attribute 'OPC.UA.DA' := '0'}
	_openValve : BOOL;
	{attribute 'OPC.UA.DA' := '0'}
	_enableStaticEliminationInterruptCmd : BOOL;
	{attribute 'OPC.UA.DA' := '0'}
	_enable : BOOL;
	{attribute 'OPC.UA.DA' := '0'}			  		   
	_raisePropertiesCmd : BOOL;	 
			
	{endregion}		 
	
	{attribute 'OPC.UA.DA' := '0'}
	_deliverMessages : INT;	
		 	
	AlarmMsg : STRING(255);
	AirValveIsOpenMsg : STRING(255);
	StaticEliminationInterruptMsg : STRING(255);
	RefreshingMsg : STRING(255);
	
	{attribute 'OPC.UA.DA' := '0'}
	message : STRING;
	
	{attribute 'OPC.UA.DA' := '0'}
	_itemScheduler : INT;
	{attribute 'OPC.UA.DA' := '0'}
	_itemRaisedProperties : INT;			
	{attribute 'OPC.UA.DA' := '0'}
	_pulseGenerator : TON;	
	
	{attribute 'OPC.UA.DA' := '0'}
	tmpConcat1 : STRING;
	{attribute 'OPC.UA.DA' := '0'}
	tmpConcat2 : STRING;
	{attribute 'OPC.UA.DA' := '0'}
	tmpConcatName : STRING; 
	{attribute 'OPC.UA.DA' := '0'}
	tmpConcatDescription : STRING;
	{attribute 'OPC.UA.DA' := '0'}
	tmpConcatAlarmID : STRING;	
	{attribute 'OPC.UA.DA' := '0'}
	_alarmCount : UINT;
	
	
END_VAR

SUPER^();

// Init device
InitDevice();

CASE _deliverMessages OF	
	EFeedbackMsgSJH108.AlarmMsg :
		AlarmMsg := message;
	EFeedbackMsgSJH108.AirValveIsOpenMsg :
		AirValveIsOpenMsg := TO_STRING(IoSJH108A.OutputOpenAirValve);
END_CASE
		
// Commands		
OpensAirValve(_openAirValveCmd, _openValve);
EnableStaticEliminationInterrupt(_enableStaticEliminationInterruptCmd, _enable);
RaisePropertiesChanged(_raisePropertiesCmd);

IF (NOT _openAirValveCmd AND NOT _enableStaticEliminationInterruptCmd AND NOT _raisePropertiesCmd) THEN	
	MessageScheduler();
END_IF

{attribute 'TcRpcEnable' := '1'}
METHOD PRIVATE EnableStaticEliminationInterrupt
VAR_INPUT
	Execute : BOOL;
	Enable : BOOL;
END_VAR
IF Execute THEN		
	_enable := Enable;
	_logger.Information(_message.Reset().Append(_config.Name).Append(' - EnableStaticEliminationInterrupt=').Append(TO_STRING(_enable)).ToString());
		
	IoSJH108A.OutputStaticEliminationInterrupt := _enable;
	_enableStaticEliminationInterruptCmd := FALSE;		
END_IF
END_METHOD

METHOD FB_init : BOOL
VAR_INPUT
	bInitRetains : BOOL; // if TRUE, the retain variables are initialized (warm start / cold start)
	bInCopyCode : BOOL;  // if TRUE, the instance afterwards gets moved into the copy code (online change)
	Config : SJH108IonizerConfig;
END_VAR
IF Config.IsEnabled THEN
	_config := Config;
	
	SUPER^._ionizerConfig.Name := Config.Name;
	SUPER^._ionizerConfig.DeviceID := Config.DeviceID;
	SUPER^._ionizerConfig.IsEnabled := Config.IsEnabled;
	SUPER^._ionizerConfig.LogLevel := Config.LogLevel;
	
	SUPER^.Name := Config.Name;
	SUPER^.DeviceID := Config.DeviceID;	
	THIS^.Family := DeviceFamily.Ionizer;
		
	IoSJH108A.OutputOpenAirValve := TRUE;
	
	_Logger.Information(_message.Reset().Append('Init ').
							Append('{').Append(TO_STRING(THIS^.Family)).Append('} - ').
							Append('{').Append(TO_STRING(Config.Name)).Append('}').ToString());																													
END_IF
END_METHOD

METHOD InitDevice
VAR_INPUT
END_VAR
IF NOT _initDevice THEN	
	_logger.Information(_message.Reset().Append(_config.Name).Append(' - Init device').ToString());
	
	THIS^.SetDone();	
	_initDevice := TRUE;	
END_IF
END_METHOD

METHOD MessageScheduler
VAR_INPUT
END_VAR
IF _pulseGenerator.Q THEN
	_pulseGenerator(IN := FALSE, PT := T#10MS);
	
	message := ' ';
	CASE _itemScheduler OF			
		0:  AirValveIsOpenMsg := ' ';
			_itemScheduler := 1;
			
		1:	ReadAlarm(); 
			_itemScheduler := 0;
	END_CASE
ELSE
	_pulseGenerator(IN := TRUE, PT := T#100MS);		
END_IF
END_METHOD

{attribute 'TcRpcEnable' := '1'}
METHOD PRIVATE OpensAirValve
VAR_INPUT
	Execute : BOOL;
	OpenValve : BOOL;
END_VAR
IF Execute THEN	
	_openValve := OpenValve;	
	_logger.Information(_message.Reset().Append(_config.Name).Append(' - Open=').Append(TO_STRING(_openValve)).ToString());
	
	IoSJH108A.OutputOpenAirValve := _openValve;
	
	_openAirValveCmd := FALSE;		
END_IF
END_METHOD

{attribute 'TcRpcEnable' := '1'}
METHOD RaisePropertiesChanged
VAR_INPUT
	Execute : BOOL;
END_VAR
IF Execute THEN		
	_raisePropertiesCmd := TRUE;	
	
	IF _pulseGenerator.Q THEN
		_pulseGenerator(IN := FALSE, PT := T#10MS);
		
		CASE _itemRaisedProperties OF		
			0:  RefreshingMsg := TO_STRING(TRUE);
				_alarmCount := 0;
				_itemRaisedProperties := 1;
				
			1: 	ReadAlarm();
				_alarmCount := _alarmCount + 1;
				IF _alarmCount = IonizerConst.NUMBER_ALARMS THEN
					_itemRaisedProperties := 2;
				END_IF							
			
			2:  RefreshingMsg := TO_STRING(FALSE);
				_raisePropertiesCmd := FALSE;
				_itemRaisedProperties := 0;		
		END_CASE	
	ELSE
		_pulseGenerator(IN := TRUE, PT := T#100MS);	
	END_IF
END_IF
END_METHOD

METHOD ReadAlarm
VAR_INPUT
END_VAR
VAR
	triggered : BOOL;
END_VAR
_deliverMessages := EFeedbackMsgSJH108.AlarmMsg;

_alarmCount := 0;

tmpConcatName := CONCAT(_config.IonizerAlarm[_alarmCount].Name, ';');
tmpConcatDescription := CONCAT(_config.IonizerAlarm[_alarmCount].Description, ';');
tmpConcatAlarmID := CONCAT(UINT_TO_STRING(_config.IonizerAlarm[_alarmCount].AlarmID), ';');

tmpConcat1 := CONCAT(tmpConcatName, tmpConcatDescription);
tmpConcat2 := CONCAT(tmpConcat1, tmpConcatAlarmID);

IF _config.IonizerAlarm[_alarmCount].Triggered THEN
	triggered := FALSE;
ELSE
	triggered := TRUE;
END_IF

message := CONCAT(tmpConcat2, TO_STRING(triggered));
END_METHOD

END_FUNCTION_BLOCK

// ---- PMShared/Hardware/Devices/Ionizers/IonizerBase.TcPOU
FUNCTION_BLOCK ABSTRACT IonizerBase EXTENDS TExecution IMPLEMENTS IDevice
VAR_INPUT
END_VAR
VAR_OUTPUT
END_VAR
VAR
	{attribute 'OPC.UA.DA' := '0'}
	_name : STRING;
	{attribute 'OPC.UA.DA' := '0'}
	_deviceID : STRING;				
	{attribute 'OPC.UA.DA' := '0'}
	_family : DeviceFamily := DeviceFamily.Ionizer;		
	{attribute 'OPC.UA.DA' := '0'}
	_logger : Logger;
	{attribute 'OPC.UA.DA' := '0'}
	_message : StringBuilder;
	{attribute 'OPC.UA.DA' := '0'}
	_ionizerConfig : DeviceConfiguration;
		
	{attribute 'OPC.UA.DA' := '0'}
	_lifeTimeCount : UINT;
	{attribute 'OPC.UA.DA' := '0'}
	_notifyIsAlive : BOOL;
	{attribute 'OPC.UA.DA' := '0'}
	_pulseIsAliveGenerator : TON;

	StateMsg : STRING(255);
	IsAliveMsg : STRING(255);
END_VAR

// Check if it's still alive	
IF _notifyIsAlive THEN
	IsAliveMsg := TO_STRING(_lifeTimeCount);
	_notifyIsAlive := FALSE;
END_IF

IF HardwareGlobalVariables.IonizerState <> State THEN
	HardwareGlobalVariables.IonizerState := State;
	StateMsg := ANY_TO_STRING(State);		
END_IF

PROPERTY DeviceID : STRING
GET
DeviceID := _deviceID;
END_GET
SET
_deviceID := DeviceID;
END_SET
END_PROPERTY

PROPERTY Family : DeviceFamily
GET
Family := _family;
END_GET
SET
_family := Family;
END_SET
END_PROPERTY

METHOD PROTECTED IsAlive
VAR_INPUT
END_VAR
_notifyIsAlive := TRUE;

IF _lifeTimeCount < 5 THEN
	_lifeTimeCount := _lifeTimeCount + 1;
ELSE
	_lifeTimeCount := 1;
END_IF
END_METHOD

PROPERTY Name : STRING
GET
Name := _name;
END_GET
SET
_name := Name;
END_SET
END_PROPERTY

END_FUNCTION_BLOCK

// ---- Service/PMs/Nst/Communication/RS232/NstBkgrdLsSerialCom.TcPOU
PROGRAM NstBkgrdLsSerialCom
VAR_INPUT
	Config : NstConfig;
END_VAR
VAR
END_VAR

// AttenuationFilterConfigs
IF Config.AttenuationFilterConfigs.FW212CAttenuationFilterConfig.IsEnabled OR 
   Config.AttenuationFilterConfigs.ELL14kAttenuationFilterConfig.IsEnabled OR 
   Config.AttenuationFilterConfigs.ELL9AttenuationFilterConfig.IsEnabled THEN
	BkgrdSerialAttenuation();	
END_IF

// LaserConfigs
IF Config.LaserConfigs.SMD12LaserConfig.IsEnabled OR 
   Config.LaserConfigs.Piano450LaserConfig.IsEnabled THEN
	BkgrdSerialLaser();
END_IF

END_PROGRAM

// ---- Service/PMs/PhotoLum/PhotoLum.TcPOU
FUNCTION_BLOCK PhotoLum EXTENDS PlcModule
VAR_INPUT
	Safety : Safety;
	
	{attribute 'OPC.UA.DA' := '0'}
	PhotoLumConfig : PhotoLumConfig;
		
	(* Chamber *)
	Chamber : PhotoLumChamber(Config := PhotoLumConfig.ChamberConfigs.PhotoLumChamberConfig);
			
	(* Chuck *)
	Chuck : PhotoLumChuck(Config := PhotoLumConfig.ChuckConfigs.PhotoLumChuckConfig);
	
	(* Axes *)
	Ps10Axis : Ps10Axis(Config := PhotoLumConfig.AxesConfigs.Ps10OwisAxisConfig); 
		
	(* Lights *)
	EvosensLight : EvosensLight(Config := PhotoLumConfig.LightConfigs.EvosensLightConfig);
	ArduinoLight : ArduinoLight(Config := PhotoLumConfig.LightConfigs.ArduinoLightConfig);
	
	(* DistanceSensorConfigs *) 
	MicroEpsilonDistanceSensor : MicroEpsilonDistanceSensor(Config := PhotoLumConfig.DistanceSensorConfigs.MicroEpsilonDistanceSensorConfig);
	
	//{attribute 'OPC.UA.DA' := '0'}
	//EfemInterlockArmExtendedEnable AT %Q* : BOOL;
END_VAR
VAR_OUTPUT
END_VAR
VAR
END_VAR


SUPER^();

IF PhotoLumConfig.SafetyIsEnabled THEN
	Safety();
END_IF

IF PhotoLumConfig.ChamberConfigs.PhotoLumChamberConfig.IsEnabled THEN
	Chamber();	
END_IF

IF PhotoLumConfig.ChuckConfigs.PhotoLumChuckConfig.IsEnabled THEN
	Chuck();		
END_IF

IF PhotoLumConfig.AxesConfigs.Ps10OwisAxisConfig.IsEnabled THEN
	Ps10Axis();	
END_IF

(* Lights *)
IF PhotoLumConfig.LightConfigs.EvosensLightConfig.IsEnabled THEN
	EvosensLight();
	IF EvosensLight.InitConfigSerialCom THEN
		;
	END_IF
ELSIF PhotoLumConfig.LightConfigs.ArduinoLightConfig.IsEnabled THEN
	ArduinoLight();
	IF ArduinoLight.InitConfigSerialCom THEN
		;
	END_IF
END_IF

IF PhotoLumConfig.DistanceSensorConfigs.MicroEpsilonDistanceSensorConfig.IsEnabled THEN
	MicroEpsilonDistanceSensor();	
END_IF


// Conditions for authorising the arm to enter the chamber
//
// Attention : bien mettre le loading position en fonction du diametre wafer
// Pour l'instant bloquer l'info à transmettre au robot
IF Chamber.SlitDoorPosition = ESlitDoorPosition.Open (*AND 
   Chamber.IsInLoadingPosition = TRUE *) THEN	
	//EfemInterlockArmExtendedEnable := TRUE;
ELSE
	//EfemInterlockArmExtendedEnable := FALSE;
END_IF

METHOD FB_init : BOOL
VAR_INPUT
	bInitRetains : BOOL; // if TRUE, the retain variables are initialized (warm start / cold start)
	bInCopyCode : BOOL;  // if TRUE, the instance afterwards gets moved into the copy code (online change)
	Config : PhotoLumConfig;
END_VAR
PhotoLumConfig := Config;
PhotoLumBkgrdSerialCom(Config := PhotoLumConfig);

IF Config.IsEnabled THEN
	_logger.Information('Photolum devices initialization starting...');
END_IF	

